// TIA Portal project "Blister 080520_V16_1" (V16)

(* hardware
DEVICE "S7-1200 station_1"  S7-1200 Station
   slot 0: "Rack_0"  S7-1200 Rack  Rack  V1.0
   slot 1: "PLC_1"  CPU 1215C DC/DC/DC  6ES7 215-1AG40-0XB0  V4.2
DEVICE "PC-System_1"  SIMATIC PC station
   slot 0: "SIMATIC PC station"  Rail  SIMATIC PC-Station  V1.0
      slot 125: "Stationmanager"  Station_Manager  V6.0.4
   slot 1: "HMI_RT_1"  WinCC RT Advanced  6AV2 104-0xxxx-xxxx  15.0.0.0
      slot 33792: "Host interface"  Host interface
   slot 2: "IE general_1"  IE General  IE_CP  V8.2.0
*)

// ===== PLC "PLC_1"  CPU 1215C DC/DC/DC =====

VAR_GLOBAL   // PLC tag table "Default tag table"
   "System_Byte" AT %MB1000 : Byte;
   "FirstScan" AT %M1000.0 : Bool;
   "DiagStatusUpdate" AT %M1000.1 : Bool;
   "AlwaysTRUE" AT %M1000.2 : Bool;
   "AlwaysFALSE" AT %M1000.3 : Bool;
   "Clock_Byte" AT %MB1001 : Byte;
   "Clock_10Hz" AT %M1001.0 : Bool;
   "Clock_5Hz" AT %M1001.1 : Bool;
   "Clock_2.5Hz" AT %M1001.2 : Bool;
   "Clock_2Hz" AT %M1001.3 : Bool;
   "Clock_1.25Hz" AT %M1001.4 : Bool;
   "Clock_1Hz" AT %M1001.5 : Bool;
   "Clock_0.625Hz" AT %M1001.6 : Bool;
   "Clock_0.5Hz" AT %M1001.7 : Bool;
   "System_Byte(1)" AT %MB1000 : Byte;
   "point_1" AT %M0.0 : Bool;
   "point_2" AT %M0.1 : Bool;
   "a" AT %MD2 : Real;
   "e" AT %MD6 : Real;
   "g" AT %MD10 : Real;
   "ii" AT %MD14 : Real;
   "oo" AT %MD18 : Real;
   "pp" AT %MD22 : Real;
   "rr" AT %MD26 : Real;
   "Run" AT %M0.2 : Bool;
   "Shift" AT %M0.3 : Bool;
   "Trig_2" AT %M0.4 : Bool;
   "Enable" AT %M0.5 : Bool;
   "Timer_Main" AT %MD30 : Time;
   "Angle" AT %MW34 : Int;
   "Temp_1" AT %MD44 : Real;
   "Forming_Trig" AT %M0.6 : Bool;
   "Forming_Enable" AT %M0.7 : Bool;
   "Servo_Pull_Enable" AT %M1.0 : Bool;
   "Servo_Pull_CCW_Trig" AT %M1.1 : Bool;
   "Servo_Pull_CW_Trig" AT %M1.2 : Bool;
   "PinHole_Detect" AT %M1.3 : Bool;
   "Trig3" AT %M1.4 : Bool;
   "PinHole_Write" AT %M1.5 : Bool;
   "T_Simu_Angle" AT %MW36 : Int;
   "Simu_Angle_2" AT %MD38 : Time;
   "Trig4" AT %M1.6 : Bool;
   "Trig5" AT %M1.7 : Bool;
   "Reset_C" AT %M42.0 : Bool;
   "Trig6" AT %M42.1 : Bool;
   "Step" AT %MW52 : Int;
   "EN_Feed_1_Step" AT %M42.2 : Bool;
   "Feeder_Enough_Step" AT %M42.3 : Bool;
   "Trig8" AT %M42.4 : Bool;
   "Set" AT %M42.5 : Bool;
   "Trig9" AT %M42.6 : Bool;
   "Do" AT %M42.7 : Bool;
   "Trig11" AT %M43.0 : Bool;
   "trig12" AT %M43.1 : Bool;
   "Feeder_Trig" AT %M43.2 : Bool;
   "Feeder_Enough_Angle" AT %M43.3 : Bool;
   "Step_Calcu" AT %MW48 : Int;
   "Trig13" AT %M43.4 : Bool;
   "Pull_2" AT %M43.5 : Bool;
   "trig14" AT %M43.6 : Bool;
   "trig15" AT %M43.7 : Bool;
   "trig16" AT %M50.0 : Bool;
   "Ghi" AT %M50.1 : Bool;
   "Ghi2" AT %M50.2 : Bool;
   "Write_not_feed" AT %M50.3 : Bool;
   "Trig17" AT %M50.4 : Bool;
   "Write_not_feed_2" AT %M50.5 : Bool;
   "trig18" AT %M50.6 : Bool;
   "Write_feed_ok" AT %M50.7 : Bool;
   "Write_not_feed_3" AT %M51.0 : Bool;
   "test" AT %M51.1 : Bool;
   "testmw" AT %MB54 : Byte;
END_VAR

DATA_BLOCK "Forming_Aplice_DB"   // DB9
{ S7_Optimized_Access := 'TRUE' }
VERSION : 0.1
// stored: InstanceOfName Forming_Aplice
"Forming_Aplice"
BEGIN
END_DATA_BLOCK

DATA_BLOCK "Blister_Animation"   // DB10
{ S7_Optimized_Access := 'TRUE' }
VERSION : 0.1
   VAR
      Blister_1 : Array[0..50] of Word;
      Blister_Matrix : Array[0..50] of Word;
   END_VAR
BEGIN
END_DATA_BLOCK

DATA_BLOCK "Blister_Show"   // DB11
{ S7_Optimized_Access := 'TRUE' }
VERSION : 0.1
   VAR RETAIN
      Total_Row : Int := 6;
      Total_Blister_Column : Int := 20;
   END_VAR
   VAR
      Total_Blister_Column_Temp : Int := 20;
      Arr : Array[0..10] of Int;
   END_VAR
BEGIN
END_DATA_BLOCK

DATA_BLOCK "Shift_Blister_DB"   // DB12
{ S7_Optimized_Access := 'TRUE' }
VERSION : 0.1
// stored: InstanceOfName Shift_Blister
"Shift_Blister"
BEGIN
END_DATA_BLOCK

DATA_BLOCK "Station_Position"   // DB13
{ S7_Optimized_Access := 'TRUE' }
VERSION : 0.1
   VAR
      Cut_to_ApliceALU : Int := 5;
      Cut_to_Camera : Int := 8;
      Cut_to_Matrix_Feeder : Int := 11;
      Cut_to_PinHole : Int := 14;
      Cut_to_Forming : Int := 17;
   END_VAR
BEGIN
END_DATA_BLOCK

DATA_BLOCK "Machine_Data"   // DB14
{ S7_Optimized_Access := 'TRUE' }
VERSION : 0.1
   VAR RETAIN
      Angle : Int;
      Length_Step : Int := 83;
      SV_Machine_Speed : Int := 30;
   END_VAR
BEGIN
END_DATA_BLOCK

DATA_BLOCK "Matrix_Feeder_DB"   // DB15
{ S7_Optimized_Access := 'TRUE' }
VERSION : 0.1
// stored: InstanceOfName Matrix_Feeder
"Matrix_Feeder"
BEGIN
END_DATA_BLOCK

DATA_BLOCK "Write_Blister_Animation_DB"   // DB17
{ S7_Optimized_Access := 'TRUE' }
VERSION : 0.1
// stored: InstanceOfName Write_Blister_Animation
"Write_Blister_Animation"
BEGIN
END_DATA_BLOCK

DATA_BLOCK "Forming_Module_DB"   // DB20
{ S7_Optimized_Access := 'TRUE' }
VERSION : 0.1
// stored: InstanceOfName Forming_Module
"Forming_Module"
BEGIN
END_DATA_BLOCK

DATA_BLOCK "Batch_Management_DB"   // DB22
{ S7_Optimized_Access := 'TRUE' }
VERSION : 0.1
// stored: InstanceOfName Batch_Management
"Batch_Management"
BEGIN
   Lot_Size := 500;
   SV_Sampling_Time := 1;
   Q_Reset_New_Lot := TRUE;
   Reset_Sampling_Time := TRUE;
   C1.QD := TRUE;
   C1.PV := 100000;
   T_Sampling_Time_1.ST := T#52M_54S_448MS;
   T_Sampling_Time_2.ST := T#52M_54S_448MS;
   T.ST := T#52M_54S_448MS;
   T.PT := T#1M_40S;
END_DATA_BLOCK

DATA_BLOCK "Total_Time_Run_DB"   // DB23
{ S7_Optimized_Access := 'TRUE' }
VERSION : 0.1
// stored: InstanceOfName Total_Time_Run
"Total_Time_Run"
BEGIN
END_DATA_BLOCK

DATA_BLOCK "Recipe_Data"   // DB24
{ S7_Optimized_Access := 'TRUE' }
VERSION : 0.1
   VAR RETAIN
      Data_1 : Int;
      Data_2 : Int;
      Data_3 : Int;
      Data_4 : Int;
      Data_5 : Int;
   END_VAR
BEGIN
END_DATA_BLOCK

DATA_BLOCK "Batch_Data"   // DB25
{ S7_Optimized_Access := 'TRUE' }
VERSION : 0.1
   VAR RETAIN
      Time_Start : DTL;
      Time_Stop : DTL;
   END_VAR
BEGIN
END_DATA_BLOCK

// folder: DB_of_FB

DATA_BLOCK "Calib_Speed_DB"   // DB1
{ S7_Optimized_Access := 'TRUE' }
VERSION : 0.1
// stored: InstanceOfName Calib_Speed_Output
"Calib_Speed_Output"
BEGIN
END_DATA_BLOCK

DATA_BLOCK "Scale_Analog_DB"   // DB3
{ S7_Optimized_Access := 'TRUE' }
VERSION : 0.1
// stored: InstanceOfName Scale_Analog_Output
"Scale_Analog_Output"
BEGIN
END_DATA_BLOCK

DATA_BLOCK "Scale_Analog_Input_DB"   // DB4
{ S7_Optimized_Access := 'TRUE' }
VERSION : 0.1
// stored: InstanceOfName Scale_Analog_Input
"Scale_Analog_Input"
BEGIN
END_DATA_BLOCK

DATA_BLOCK "Calib_Temperature_Input_DB"   // DB5
{ S7_Optimized_Access := 'TRUE' }
VERSION : 0.1
// stored: InstanceOfName Calib_Temperature_Input
"Calib_Temperature_Input"
BEGIN
END_DATA_BLOCK

// folder: Main_program/Conveyor

DATA_BLOCK "Conveyor"   // DB2
{ S7_Optimized_Access := 'TRUE' }
VERSION : 0.1
   VAR
      Calib_Enable : Bool;
      B_Calib_Dim_Point_1 : Bool;
      B_Calib_Dim_Point_2 : Bool;
      SV_Calib_Speed_Point_1 : Int;
      SV_Calib_Speed_Point_2 : Int;
   END_VAR
   VAR RETAIN
      Calib_Range_Analog_Low : Int;
      Calib_Range_Analog_High : Int;
      Calib_Range_Speed_Low : Int;
      Calib_Range_Speed_High : Int;
   END_VAR
   VAR
      SV_Speed : Int;
      O_Analog : Int;
      B_RunConveyor_Speed_Min : Bool;
      B_RunConveyor_Speed_Max : Bool;
      B_Calib_OK : Bool;
      B_Calib_Default : Bool;
      O_Calib_Result : Bool;
      O_Run : Bool;
      H_PID_State : Int;
      H_Stop_Kp : Real;
      H_Stop_Ki : Real;
      H_Stop_Kd : Real;
      H_Run_Kp : Real;
      H_Run_Ki : Real;
      H_Run_Kd : Real;
      B_PID_Default : Bool;
      Stop_Kp_1 : Real;
      Stop_Ki_1 : Real;
      Stop_Kd_1 : Real;
      Run_Kp_1 : Real;
      Run_Ki_1 : Real;
      Run_Kd_1 : Real;
   END_VAR
BEGIN
END_DATA_BLOCK

DATA_BLOCK "PID Setting_DB"   // DB8
{ S7_Optimized_Access := 'TRUE' }
VERSION : 0.1
// stored: InstanceOfName PID Setting
"PID Setting"
BEGIN
END_DATA_BLOCK

// folder: Main_program/Temperature_Top

DATA_BLOCK "Temperature_Top"   // DB6
{ S7_Optimized_Access := 'TRUE' }
VERSION : 0.1
   VAR
      Calib_Enable : Bool;
      B_Calib_Dim_Point_1 : Bool;
      B_Calib_Dim_Point_2 : Bool;
   END_VAR
   VAR RETAIN
      O_Calib_Range_Analog_Min : Int;
      O_Calib_Range_Analog_Max : Int;
      O_Calib_Range_Temper_Min : Int;
      O_Calib_Range_Temper_Max : Int;
   END_VAR
   VAR
      PV_Temper : Int;
      B_Calib_OK : Bool;
      B_Default : Bool;
      I_Analog_Read : Int;
      B_Default_3 : Bool;
      Calib_Result : Bool;
      SV_Point_1_Temper : Int;
      SV_Point_2_Temper : Int;
      SV_Temper : Int;
      PWM_Out : Bool;
   END_VAR
BEGIN
END_DATA_BLOCK

// folder: System blocks/Program resources

DATA_BLOCK "IEC_Timer_0_DB"   // DB16
{ S7_Optimized_Access := 'TRUE' }
AUTHOR : Simatic
FAMILY : IEC
NAME : IEC_TMR
VERSION : 1.0
// stored: InstanceOfName IEC_TIMER
"IEC_TIMER"
BEGIN
END_DATA_BLOCK

DATA_BLOCK "IEC_Timer_0_DB_1"   // DB18
{ S7_Optimized_Access := 'TRUE' }
AUTHOR : Simatic
FAMILY : IEC
NAME : IEC_TMR
VERSION : 1.0
// stored: InstanceOfName IEC_TIMER
"IEC_TIMER"
BEGIN
END_DATA_BLOCK

DATA_BLOCK "IEC_Timer_0_DB_2"   // DB19
{ S7_Optimized_Access := 'TRUE' }
AUTHOR : Simatic
FAMILY : IEC
NAME : IEC_TMR
VERSION : 1.0
// stored: InstanceOfName IEC_TIMER
"IEC_TIMER"
BEGIN
END_DATA_BLOCK

DATA_BLOCK "IEC_Timer_0_DB_3"   // DB21
{ S7_Optimized_Access := 'TRUE' }
AUTHOR : Simatic
FAMILY : IEC
NAME : IEC_TMR
VERSION : 1.0
// stored: InstanceOfName IEC_TIMER
"IEC_TIMER"
BEGIN
END_DATA_BLOCK

// folder: (top level)

FUNCTION_BLOCK "Forming_Aplice"   // FB6, LAD
{ S7_Optimized_Access := 'TRUE' }
VERSION : 0.1
   VAR_INPUT
      Sensor : Bool;
   END_VAR
BEGIN

REGION Network 1
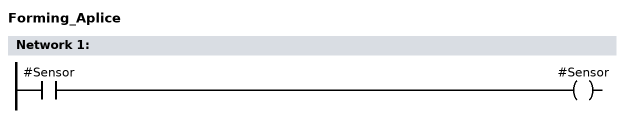
   RUNG wire#powerrail
      Contact( #Sensor )
      Coil( #Sensor )
   END_RUNG
   // the same network as SCL:
   #Sensor := #Sensor;
END_REGION
END_FUNCTION_BLOCK

FUNCTION_BLOCK "Shift_Blister"   // FB7, LAD
{ S7_Optimized_Access := 'TRUE' }
VERSION : 0.1
   VAR_INPUT
      Number_Column : Int;
   END_VAR
   VAR_IN_OUT
      Trig : Bool;
   END_VAR
   VAR
      i : Int;
   END_VAR
BEGIN

REGION Network 2 (SCL)
   IF #Trig = TRUE THEN
       "Blister_Animation".Blister_1[#Number_Column + 1] := 0;
       FOR #i := 0 TO #Number_Column DO
           "Blister_Animation".Blister_1[#i] := "Blister_Animation".Blister_1[#i + 1];
           "Blister_Animation".Blister_Matrix[#i] := "Blister_Animation".Blister_Matrix[#i + 1];
       END_FOR;
       #Trig := FALSE;
       // #Do := FALSE;
   END_IF;
END_REGION
END_FUNCTION_BLOCK

FUNCTION_BLOCK "Matrix_Feeder"   // FB8, LAD
{ S7_Optimized_Access := 'TRUE' }
VERSION : 0.1
   VAR_INPUT
      Angel_Machine : Int;
      Pull_Trig : Bool;
      "Switch_on/off" : Bool;
   END_VAR
   VAR_OUTPUT
      Q_Feeder : Bool;
   END_VAR
   VAR
      Counte : IEC_COUNTER;
   END_VAR
   VAR RETAIN
      Feed_1_Step : Bool;
      EN_Feed_2_Step : Bool;
   END_VAR
   VAR
      Feed_2_Step : Bool;
      Angel_Begin : Int := 170;
      Angel_End : Int := 210;
      Angel_Begin_Offset : Int;
      I_Step_Feeder : Int := 1;
      Trig1 : Bool;
   END_VAR
   VAR_TEMP   // added for the SCL form of the ladder/FBD networks
      _w1 : Bool;
      _w2 : Bool;
   END_VAR
BEGIN

REGION Network 1: Reset step feer
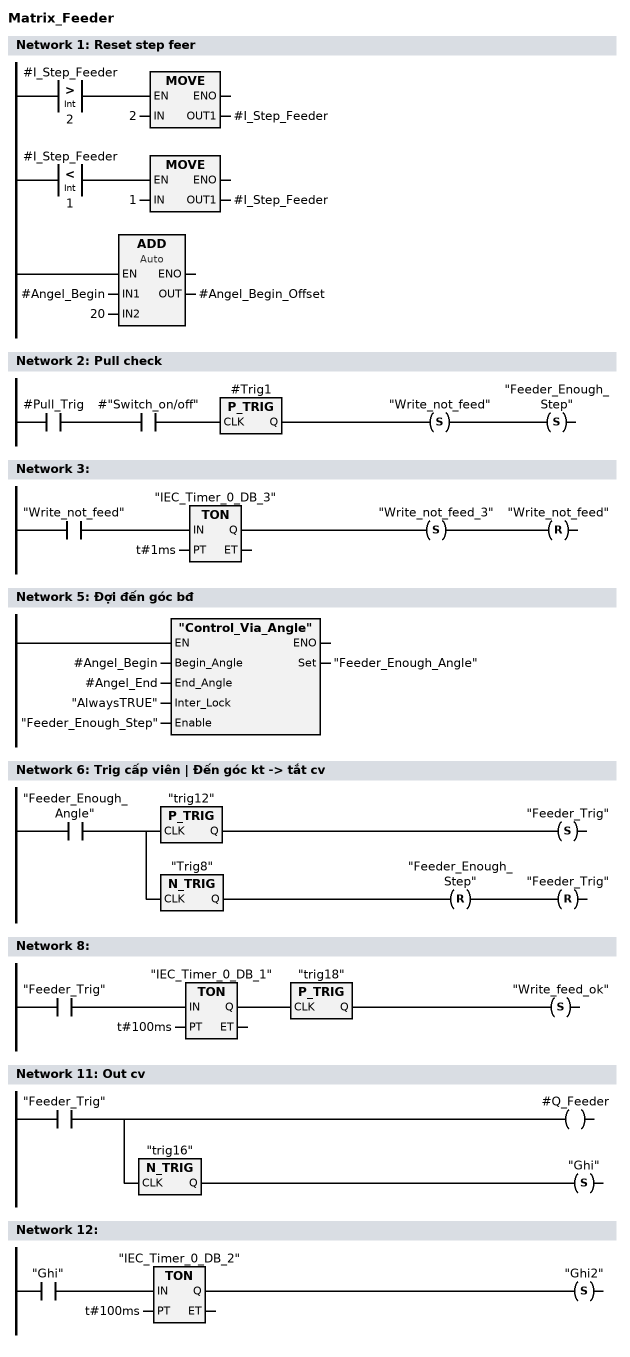
   RUNG wire#powerrail
      { S7_Templates := "SrcType := Int" } GT_Contact(in1 := #I_Step_Feeder, in2 := 2)
      Move(in := 2, out1 => #I_Step_Feeder)
   END_RUNG
   RUNG wire#powerrail
      { S7_Templates := "SrcType := Int" } LT_Contact(in1 := #I_Step_Feeder, in2 := 1)
      Move(in := 1, out1 => #I_Step_Feeder)
   END_RUNG
   RUNG wire#powerrail
      Add(in1 := #Angel_Begin, in2 := 20, out => #Angel_Begin_Offset)
   END_RUNG
   // the same network as SCL:
   IF #I_Step_Feeder > 2 THEN #I_Step_Feeder := 2; END_IF;
   IF #I_Step_Feeder < 1 THEN #I_Step_Feeder := 1; END_IF;
   #Angel_Begin_Offset := #Angel_Begin + 20;
END_REGION

REGION Network 2: Pull check
   RUNG wire#powerrail
      Contact( #Pull_Trig )
      Contact( #"Switch_on/off" )
      P_Trig( #Trig1 )
      S_Coil( "Write_not_feed" )
      S_Coil( "Feeder_Enough_Step" )
   END_RUNG
   // the same network as SCL:
   #_w1 := #Pull_Trig AND #"Switch_on/off";
   #_w2 := #_w1 AND NOT #Trig1;   // rising edge
   #Trig1 := #_w1;
   IF #_w2 THEN
       "Write_not_feed" := TRUE;
       "Feeder_Enough_Step" := TRUE;
   END_IF;
END_REGION

REGION Network 3
   "IEC_Timer_0_DB_3".TON(IN := "Write_not_feed", PT := t#1ms);
   IF "IEC_Timer_0_DB_3".Q THEN
       "Write_not_feed_3" := TRUE;
       "Write_not_feed" := FALSE;
   END_IF;
END_REGION

REGION Network 4 (SCL)
   //IF FALSE = true THEN
   IF "Write_not_feed_3" = true THEN
       //  Bước cv = 2 thi kiem tra 2 hang
       IF #I_Step_Feeder = 2 THEN
           "Blister_Animation".Blister_1["Station_Position".Cut_to_Matrix_Feeder] := 0;
           "Blister_Animation".Blister_1["Station_Position".Cut_to_Matrix_Feeder + 1] := 0;
       END_IF;
       // = 1
       IF #I_Step_Feeder = 1 THEN
           "Blister_Animation".Blister_1["Station_Position".Cut_to_Matrix_Feeder] := 0;
       END_IF;
       "Write_not_feed_3" := FALSE;
   END_IF;
END_REGION

REGION Network 5: Đợi đến góc bđ
   RUNG wire#powerrail
      "Control_Via_Angle"(Begin_Angle := #Angel_Begin, End_Angle := #Angel_End, Inter_Lock := "AlwaysTRUE", Enable := "Feeder_Enough_Step", Set => "Feeder_Enough_Angle")
   END_RUNG
   // the same network as SCL:
   "Control_Via_Angle"(Begin_Angle := #Angel_Begin,
                       End_Angle := #Angel_End,
                       Inter_Lock := "AlwaysTRUE",
                       Enable := "Feeder_Enough_Step",
                       Set => "Feeder_Enough_Angle");
END_REGION

REGION Network 6: Trig cấp viên | Đến góc kt -> tắt cv
   RUNG wire#powerrail
      Contact( "Feeder_Enough_Angle" )
      wire#w1
      P_Trig( "trig12" )
      S_Coil( "Feeder_Trig" )
   END_RUNG
   RUNG wire#w1
      N_Trig( "Trig8" )
      R_Coil( "Feeder_Enough_Step" )
      R_Coil( "Feeder_Trig" )
   END_RUNG
   // the same network as SCL:
   #_w1 := "Feeder_Enough_Angle" AND NOT "trig12";   // rising edge
   "trig12" := "Feeder_Enough_Angle";
   IF #_w1 THEN "Feeder_Trig" := TRUE; END_IF;
   #_w2 := NOT "Feeder_Enough_Angle" AND "Trig8";   // falling edge
   "Trig8" := "Feeder_Enough_Angle";
   IF #_w2 THEN
       "Feeder_Enough_Step" := FALSE;
       "Feeder_Trig" := FALSE;
   END_IF;
END_REGION

REGION Network 7 (SCL): Kiểm tra đk cv | buoc cv = 1 or 2
   //IF FALSE = true THEN
   IF "Feeder_Trig" = true THEN
      //  Bước cv = 2 thi kiem tra 2 hang
       IF #I_Step_Feeder = 2 THEN 
           IF "Blister_Animation".Blister_Matrix["Station_Position".Cut_to_Matrix_Feeder] <> 16#3F OR "Blister_Animation".Blister_Matrix["Station_Position".Cut_to_Matrix_Feeder + 1] <> 16#3F THEN
               "Feeder_Trig" := FALSE;
           END_IF;
      END_IF;
       // = 1
       IF #I_Step_Feeder = 1 THEN
           IF "Blister_Animation".Blister_Matrix["Station_Position".Cut_to_Matrix_Feeder] <> 16#3F THEN
               "Feeder_Trig" := FALSE;
               "Blister_Animation".Blister_1["Station_Position".Cut_to_Matrix_Feeder] := 0;
           END_IF;
       END_IF;
   END_IF;
END_REGION

REGION Network 8
   "IEC_Timer_0_DB_1".TON(IN := "Feeder_Trig", PT := t#100ms);
   #_w1 := "IEC_Timer_0_DB_1".Q AND NOT "trig18";   // rising edge
   "trig18" := "IEC_Timer_0_DB_1".Q;
   IF #_w1 THEN "Write_feed_ok" := TRUE; END_IF;
END_REGION

REGION Network 9 (SCL)
   //IF FALSE = true THEN
   IF "Write_feed_ok" = true THEN
       //  Bước cv = 2 thi ghi 2 hang ok sau khi qua cvmt
       IF #I_Step_Feeder = 2 THEN
           "Blister_Animation".Blister_1["Station_Position".Cut_to_Matrix_Feeder] := 16#3f;
           "Blister_Animation".Blister_1["Station_Position".Cut_to_Matrix_Feeder + 1] := 16#3f;
       END_IF;
       // = 1
       IF #I_Step_Feeder = 1 THEN
           "Blister_Animation".Blister_1["Station_Position".Cut_to_Matrix_Feeder] := 16#3f;
       END_IF;
       "Write_feed_ok" := FALSE;
   END_IF;
END_REGION

REGION Network 10 (SCL)
   IF "Write_not_feed_2" = TRUE THEN
       "Blister_Animation".Blister_1["Station_Position".Cut_to_Matrix_Feeder] := 0;
       "Blister_Animation".Blister_1["Station_Position".Cut_to_Matrix_Feeder + 1] := 0;
       ;
   "Write_not_feed_2" := FALSE;
   END_IF;
END_REGION

REGION Network 11: Out cv
   RUNG wire#powerrail
      Contact( "Feeder_Trig" )
      wire#w1
      Coil( #Q_Feeder )
   END_RUNG
   RUNG wire#w1
      N_Trig( "trig16" )
      S_Coil( "Ghi" )
   END_RUNG
   // the same network as SCL:
   #Q_Feeder := "Feeder_Trig";
   #_w1 := NOT "Feeder_Trig" AND "trig16";   // falling edge
   "trig16" := "Feeder_Trig";
   IF #_w1 THEN "Ghi" := TRUE; END_IF;
END_REGION

REGION Network 12
   "IEC_Timer_0_DB_2".TON(IN := "Ghi", PT := t#100ms);
   IF "IEC_Timer_0_DB_2".Q THEN "Ghi2" := TRUE; END_IF;
END_REGION

REGION Network 13 (SCL): Ghi gia tri 0 sau khi cap vien ok
   IF "Ghi2" = true THEN
       IF #I_Step_Feeder = 2 THEN
           "Blister_Animation".Blister_Matrix["Station_Position".Cut_to_Matrix_Feeder] := 0;
           "Blister_Animation".Blister_Matrix["Station_Position".Cut_to_Matrix_Feeder + 1] := 0;
           ;
       END_IF;
       // buoc cv = 1
       IF #I_Step_Feeder = 1 THEN
           "Blister_Animation".Blister_Matrix["Station_Position".Cut_to_Matrix_Feeder] := 0;
           ;
       END_IF;
   "Ghi" := FALSE;
   "Ghi2" := FALSE;
   END_IF;
END_REGION
END_FUNCTION_BLOCK

FUNCTION_BLOCK "Write_Blister_Animation"   // FB9, LAD
{ S7_Optimized_Access := 'TRUE' }
VERSION : 0.1
   VAR_INPUT
      Forming_Trig : Bool;
   END_VAR
   VAR
      Trig : Bool;
      Write_Forming : Bool;
   END_VAR
   VAR_TEMP   // added for the SCL form of the ladder/FBD networks
      _w1 : Bool;
   END_VAR
BEGIN

REGION Network 1
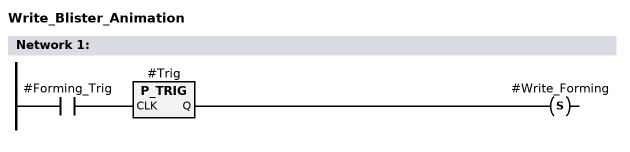
   RUNG wire#powerrail
      Contact( #Forming_Trig )
      P_Trig( #Trig )
      S_Coil( #Write_Forming )
   END_RUNG
   // the same network as SCL:
   #_w1 := #Forming_Trig AND NOT #Trig;   // rising edge
   #Trig := #Forming_Trig;
   IF #_w1 THEN #Write_Forming := TRUE; END_IF;
END_REGION

REGION Network 2 (SCL)
   IF #Write_Forming = TRUE THEN
       "Blister_Animation".Blister_1["Station_Position".Cut_to_Forming] := 2#111111;
       "Blister_Animation".Blister_Matrix["Station_Position".Cut_to_Forming] := 2#111111;
       #Write_Forming := FALSE;

   END_IF;
END_REGION
END_FUNCTION_BLOCK

FUNCTION_BLOCK "Forming_Module"   // FB10, LAD
{ S7_Optimized_Access := 'TRUE' }
VERSION : 0.1
   VAR_INPUT
      Inter_Lock : Bool;
   END_VAR
   VAR_OUTPUT
      Forming_Trig : Bool;
   END_VAR
   VAR RETAIN
      SV_Angle_Forming_Begin : Int := 160;
      SV_Angle_Forming_End : Int := 200;
   END_VAR
   VAR
      Forming_Switch : Bool;
   END_VAR
BEGIN

REGION Network 1
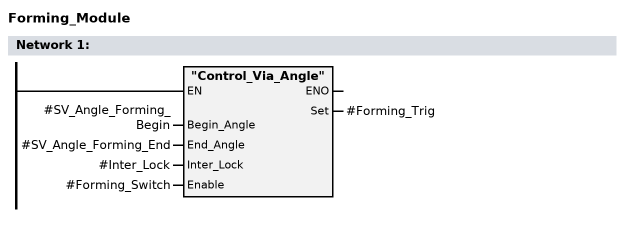
   RUNG wire#powerrail
      "Control_Via_Angle"(Begin_Angle := #SV_Angle_Forming_Begin, End_Angle := #SV_Angle_Forming_End, Enable := #Forming_Switch, Inter_Lock := #Inter_Lock, Set => #Forming_Trig)
   END_RUNG
   // the same network as SCL:
   "Control_Via_Angle"(Begin_Angle := #SV_Angle_Forming_Begin,
                       End_Angle := #SV_Angle_Forming_End,
                       Inter_Lock := #Inter_Lock,
                       Enable := #Forming_Switch,
                       Set => #Forming_Trig);
END_REGION
END_FUNCTION_BLOCK

FUNCTION_BLOCK "Batch_Management"   // FB11, LAD
{ S7_Optimized_Access := 'TRUE' }
VERSION : 0.1
   VAR_INPUT
      I_Machine_Run : Bool;
      Lot_Size : DInt;
      SV_Sampling_Time : DInt;
      Product_Name : Int;
      Batch_Number : Int;
      Batch_Size : DInt;
   END_VAR
   VAR_OUTPUT
      Q_Write_Report : Bool;
   END_VAR
   VAR_IN_OUT
      B_Start_Lot : Bool;
      B_Finish_Lot : Bool;
      B_Hold_Lot : Bool;
      Q_Reset_New_Lot : Bool;
      Reset_Sampling_Time : Bool;
      PV_Lot_Start_Time : DTL;
      PV_Lot_End_Time : DTL;
      PV_Lot_Status : USInt := 0;
      PV_Lot_Running_Total_Time : DInt;
   END_VAR
   VAR
      Trig : Bool;
      Trig2 : Bool;
      Trig3 : Bool;
      Trig4 : Bool;
      RET_VAL_1 : Int;
      RET_VAL_2 : Int;
      C1 : IEC_DCOUNTER;
   END_VAR
   VAR RETAIN
      T_Sampling_Time_1 : IEC_TIMER;
   END_VAR
   VAR
      T_Sampling_Time_2 : IEC_TIMER;
      PV_Sampling_Time : DInt;
      Trig5 : Bool;
      T : IEC_TIMER;
      Recipe_Name_1 : String;
      Recipe_Name_2 : String;
      Recipe_Record_1 : Int;
      Recipe_Record_2 : Int;
      Record_Number : Int;
   END_VAR
   VAR CONSTANT
      Running : USInt := 2;
      Finish : USInt := 0;
      Holding : USInt := 1;
   END_VAR
   VAR_TEMP   // added for the SCL form of the ladder/FBD networks
      _w1 : Bool;
      _w2 : Bool;
      _w3 : Bool;
      _w4 : Bool;
   END_VAR
BEGIN

REGION Network 1: Thời điểm bắt đầu lô
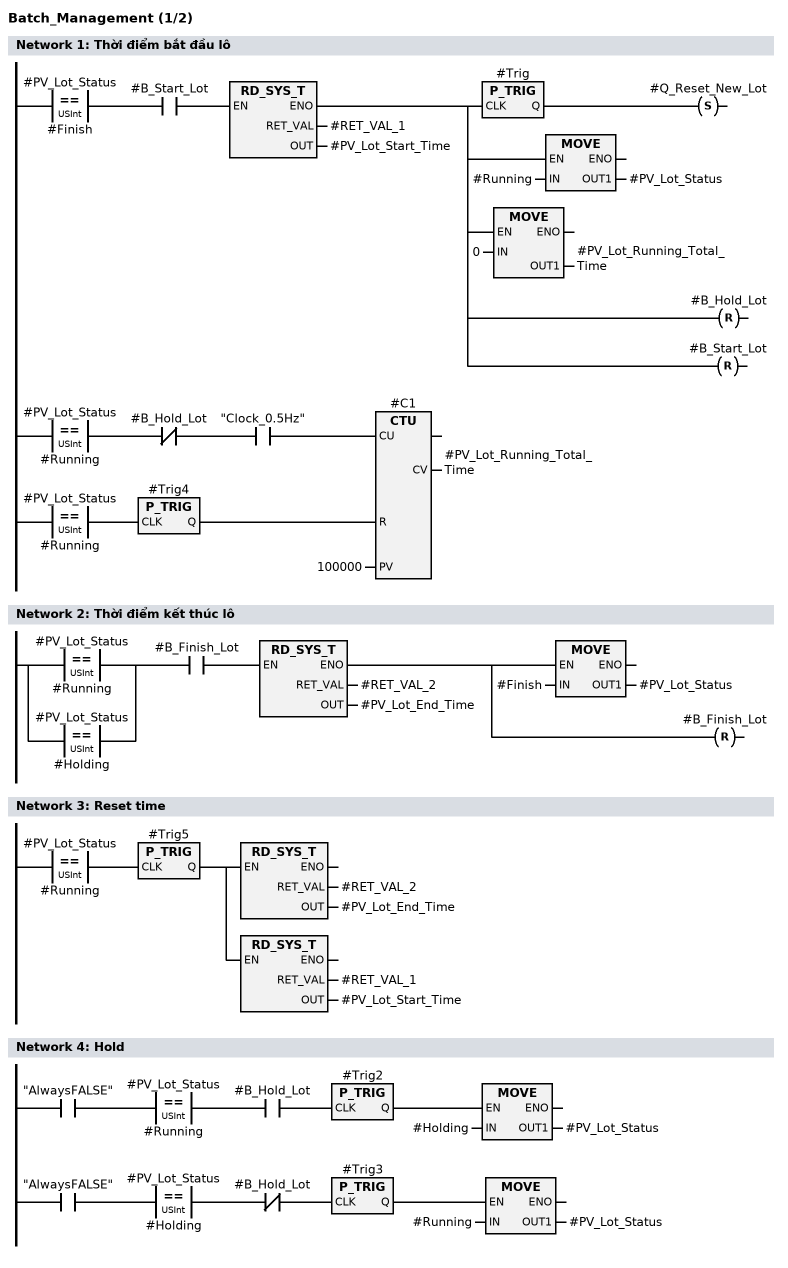
   // ENO of a box is taken as its EN; it also drops when the box reports an error
   #_w1 := (#PV_Lot_Status = #Finish) AND #B_Start_Lot;
   IF #_w1 THEN #RET_VAL_1 := RD_SYS_T(OUT => #PV_Lot_Start_Time); END_IF;
   #_w2 := #_w1 AND NOT #Trig;   // rising edge
   #Trig := #_w1;
   IF #_w2 THEN #Q_Reset_New_Lot := TRUE; END_IF;
   IF #_w1 THEN
       #PV_Lot_Status := #Running;
       #PV_Lot_Running_Total_Time := 0;
       #B_Hold_Lot := FALSE;
       #B_Start_Lot := FALSE;
   END_IF;
   #_w3 := #PV_Lot_Status = #Running;
   #_w4 := #_w3 AND NOT #Trig4;   // rising edge
   #Trig4 := #_w3;
   #C1.CTU(CU := (#PV_Lot_Status = #Running) AND NOT #B_Hold_Lot AND "Clock_0.5Hz",
           R := #_w4,
           PV := 100000,
           CV => #PV_Lot_Running_Total_Time);
END_REGION

REGION Network 2: Thời điểm kết thúc lô
   // ENO of a box is taken as its EN; it also drops when the box reports an error
   IF ((#PV_Lot_Status = #Running) OR (#PV_Lot_Status = #Holding)) AND #B_Finish_Lot THEN
       #RET_VAL_2 := RD_SYS_T(OUT => #PV_Lot_End_Time);
   END_IF;
   #_w1 := ((#PV_Lot_Status = #Running) OR (#PV_Lot_Status = #Holding)) AND #B_Finish_Lot;
   IF #_w1 THEN
       #PV_Lot_Status := #Finish;
       #B_Finish_Lot := FALSE;
   END_IF;
END_REGION

REGION Network 3: Reset time
   #_w1 := #PV_Lot_Status = #Running;
   #_w2 := #_w1 AND NOT #Trig5;   // rising edge
   #Trig5 := #_w1;
   IF #_w2 THEN
       #RET_VAL_2 := RD_SYS_T(OUT => #PV_Lot_End_Time);
       #RET_VAL_1 := RD_SYS_T(OUT => #PV_Lot_Start_Time);
   END_IF;
END_REGION

REGION Network 4: Hold
   RUNG wire#powerrail
      Contact( "AlwaysFALSE" )
      { S7_Templates := "SrcType := USInt" } EQ_Contact(in1 := #PV_Lot_Status, in2 := #Running)
      Contact( #B_Hold_Lot )
      P_Trig( #Trig2 )
      Move(in := #Holding, out1 => #PV_Lot_Status)
   END_RUNG
   RUNG wire#powerrail
      Contact( "AlwaysFALSE" )
      { S7_Templates := "SrcType := USInt" } EQ_Contact(in1 := #PV_Lot_Status, in2 := #Holding)
      I_Contact( #B_Hold_Lot )
      P_Trig( #Trig3 )
      Move(in := #Running, out1 => #PV_Lot_Status)
   END_RUNG
   // the same network as SCL:
   #_w1 := "AlwaysFALSE" AND (#PV_Lot_Status = #Running) AND #B_Hold_Lot;
   #_w2 := #_w1 AND NOT #Trig2;   // rising edge
   #Trig2 := #_w1;
   IF #_w2 THEN #PV_Lot_Status := #Holding; END_IF;
   #_w3 := "AlwaysFALSE" AND (#PV_Lot_Status = #Holding) AND NOT #B_Hold_Lot;
   #_w4 := #_w3 AND NOT #Trig3;   // rising edge
   #Trig3 := #_w3;
   IF #_w4 THEN #PV_Lot_Status := #Running; END_IF;
END_REGION

REGION Network 5: Write report
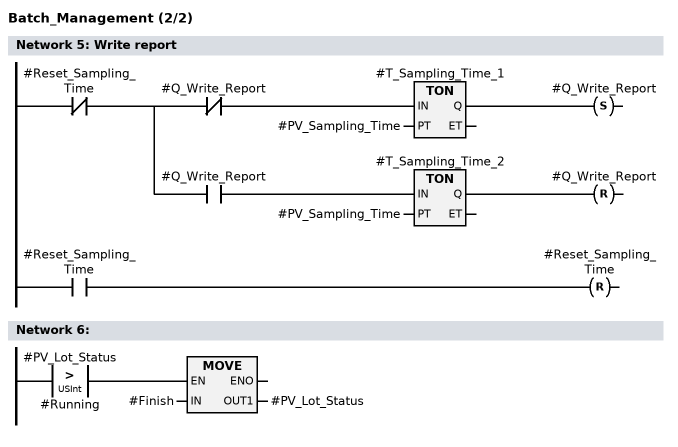
   #T_Sampling_Time_1.TON(IN := NOT #Reset_Sampling_Time AND NOT #Q_Write_Report, PT := #PV_Sampling_Time);
   IF #T_Sampling_Time_1.Q THEN #Q_Write_Report := TRUE; END_IF;
   #T_Sampling_Time_2.TON(IN := NOT #Reset_Sampling_Time AND #Q_Write_Report, PT := #PV_Sampling_Time);
   IF #T_Sampling_Time_2.Q THEN #Q_Write_Report := FALSE; END_IF;
   IF #Reset_Sampling_Time THEN #Reset_Sampling_Time := FALSE; END_IF;
END_REGION

REGION Network 6
   RUNG wire#powerrail
      { S7_Templates := "SrcType := USInt" } GT_Contact(in1 := #PV_Lot_Status, in2 := #Running)
      Move(in := #Finish, out1 => #PV_Lot_Status)
   END_RUNG
   // the same network as SCL:
   IF #PV_Lot_Status > #Running THEN #PV_Lot_Status := #Finish; END_IF;
END_REGION
END_FUNCTION_BLOCK

FUNCTION_BLOCK "Total_Time_Run"   // FB12, LAD
{ S7_Optimized_Access := 'TRUE' }
VERSION : 0.1
   VAR_OUTPUT
      "PV_Total_Time_Run_(s)" : DInt;
   END_VAR
   VAR
      C1 : IEC_DCOUNTER;
   END_VAR
BEGIN

REGION Network 1
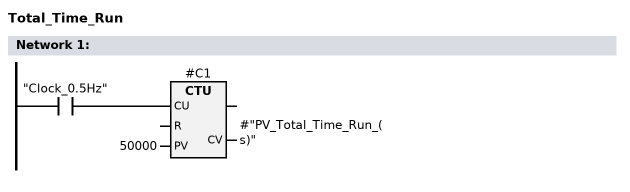
   #C1.CTU(CU := "Clock_0.5Hz", PV := 50000, CV => #"PV_Total_Time_Run_(s)");
END_REGION
END_FUNCTION_BLOCK

FUNCTION "Angle_Simu" : Void   // FC6, LAD
{ S7_Optimized_Access := 'TRUE' }
VERSION : 0.1
   VAR_TEMP
      RS : Bool;
   END_VAR
BEGIN

REGION Network 1
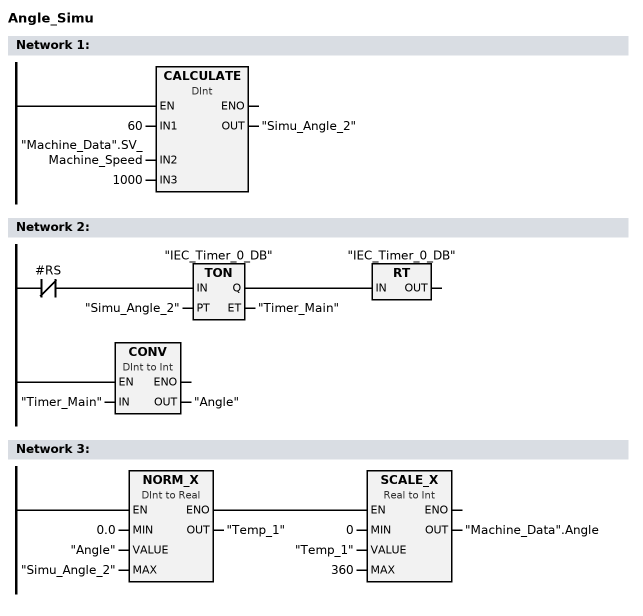
   RUNG wire#powerrail
      { S7_Templates := "SrcType := DInt"; S7_Expression := "IN1/IN2*IN3" } Calculate(in1 := 60, in2 := "Machine_Data".SV_Machine_Speed, in3 := 1000, out => "Simu_Angle_2")
   END_RUNG
   // the same network as SCL:
   "Simu_Angle_2" := 60/"Machine_Data".SV_Machine_Speed*1000;
END_REGION

REGION Network 2
   "IEC_Timer_0_DB".TON(IN := NOT #RS, PT := "Simu_Angle_2", ET => "Timer_Main");
   IF "IEC_Timer_0_DB".Q THEN RESET_TIMER("IEC_Timer_0_DB"); END_IF;
   "Angle" := DINT_TO_INT("Timer_Main");
END_REGION

REGION Network 3
   RUNG wire#powerrail
      { S7_Templates := "[SrcType := DInt, DestType := Real]" } Normalize(min := 0.0, value := "Angle", max := "Simu_Angle_2", out => "Temp_1")
      { S7_Templates := "[SrcType := Real, DestType := Int]" } Scale(min := 0, value := "Temp_1", max := 360, out => "Machine_Data".Angle)
   END_RUNG
   // the same network as SCL:
   "Temp_1" := NORM_X(MIN := 0.0, VALUE := "Angle", MAX := "Simu_Angle_2");
   "Machine_Data".Angle := SCALE_X(MIN := 0, VALUE := "Temp_1", MAX := 360);
END_REGION
END_FUNCTION

FUNCTION "Control_Via_Angle" : Void   // FC7, LAD
{ S7_Optimized_Access := 'TRUE' }
VERSION : 0.1
   VAR_INPUT
      Begin_Angle : Int;
      End_Angle : Int;
      Inter_Lock : Bool;
   END_VAR
   VAR_OUTPUT
      Set : Bool;
   END_VAR
   VAR_IN_OUT
      Enable : Bool;
   END_VAR
BEGIN

REGION Network 1
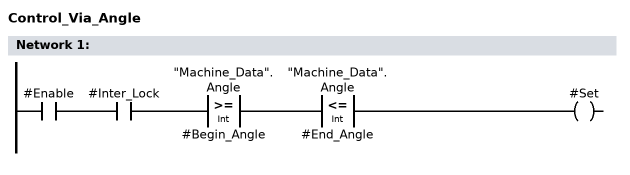
   RUNG wire#powerrail
      Contact( #Enable )
      Contact( #Inter_Lock )
      { S7_Templates := "SrcType := Int" } GE_Contact(in1 := "Machine_Data".Angle, in2 := #Begin_Angle)
      { S7_Templates := "SrcType := Int" } LE_Contact(in1 := "Machine_Data".Angle, in2 := #End_Angle)
      Coil( #Set )
   END_RUNG
   // the same network as SCL:
   #Set := #Enable AND #Inter_Lock AND ("Machine_Data".Angle >= #Begin_Angle) AND ("Machine_Data".Angle <= #End_Angle);
END_REGION
END_FUNCTION

FUNCTION "Servo_Pull" : Void   // FC8, LAD
{ S7_Optimized_Access := 'TRUE' }
VERSION : 0.1
BEGIN

REGION Network 1: CW
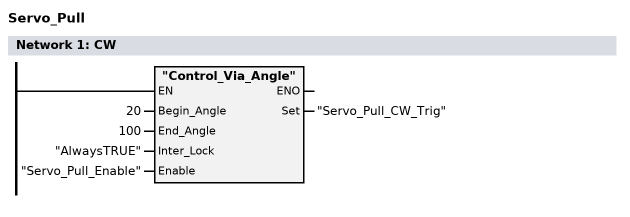
   RUNG wire#powerrail
      "Control_Via_Angle"(Begin_Angle := 20, End_Angle := 100, Inter_Lock := "AlwaysTRUE", Enable := "Servo_Pull_Enable", Set => "Servo_Pull_CW_Trig")
   END_RUNG
   // the same network as SCL:
   "Control_Via_Angle"(Begin_Angle := 20,
                       End_Angle := 100,
                       Inter_Lock := "AlwaysTRUE",
                       Enable := "Servo_Pull_Enable",
                       Set => "Servo_Pull_CW_Trig");
END_REGION
END_FUNCTION

FUNCTION "PinHole" : Void   // FC9, LAD
{ S7_Optimized_Access := 'TRUE' }
VERSION : 0.1
   VAR_TEMP   // added for the SCL form of the ladder/FBD networks
      _w1 : Bool;
      _w2 : Bool;
   END_VAR
BEGIN

REGION Network 1
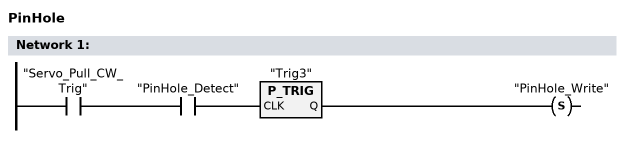
   RUNG wire#powerrail
      Contact( "Servo_Pull_CW_Trig" )
      Contact( "PinHole_Detect" )
      P_Trig( "Trig3" )
      S_Coil( "PinHole_Write" )
   END_RUNG
   // the same network as SCL:
   #_w1 := "Servo_Pull_CW_Trig" AND "PinHole_Detect";
   #_w2 := #_w1 AND NOT "Trig3";   // rising edge
   "Trig3" := #_w1;
   IF #_w2 THEN "PinHole_Write" := TRUE; END_IF;
END_REGION

REGION Network 2 (SCL)
   IF "PinHole_Write" = TRUE THEN
       "Blister_Animation".Blister_1["Station_Position".Cut_to_PinHole] := 2#000000;
       "Blister_Animation".Blister_Matrix["Station_Position".Cut_to_PinHole] := 2#000000;
       "PinHole_Write" := FALSE;

   END_IF;
END_REGION
END_FUNCTION

ORGANIZATION_BLOCK "Main"   // OB1, LAD, ProgramCycle
TITLE = "Main Program Sweep (Cycle)"
{ S7_Optimized_Access := 'TRUE' }
VERSION : 0.1
   VAR_INPUT
      Initial_Call : Bool;   // Initial call of this OB
      Remanence : Bool;   // =True, if remanent data are available
   END_VAR
   VAR_TEMP
      Trig_1 : Bool;
   END_VAR
   VAR_TEMP   // added for the SCL form of the ladder/FBD networks
      _w1 : Bool;
      _w2 : Bool;
   END_VAR
BEGIN

REGION Network 1: Conveyor
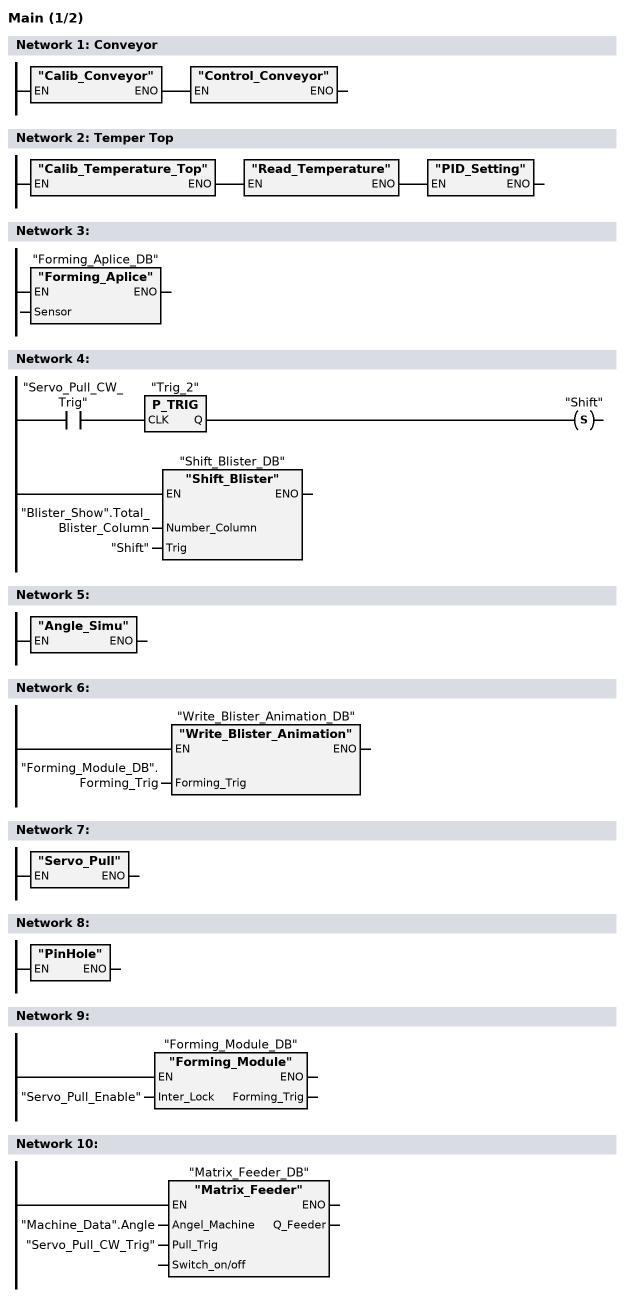
   RUNG wire#powerrail
      "Calib_Conveyor"()
      "Control_Conveyor"()
   END_RUNG
   // the same network as SCL:
   "Calib_Conveyor"(ENO => #_w1);
   IF #_w1 THEN "Control_Conveyor"(); END_IF;
END_REGION

REGION Network 2: Temper Top
   RUNG wire#powerrail
      "Calib_Temperature_Top"()
      "Read_Temperature"()
      "PID_Setting"()
   END_RUNG
   // the same network as SCL:
   "Calib_Temperature_Top"(ENO => #_w1);
   "Read_Temperature"(EN := #_w1, ENO => #_w2);
   IF #_w2 THEN "PID_Setting"(); END_IF;
END_REGION

REGION Network 3
   RUNG wire#powerrail
      "Forming_Aplice_DB"(Sensor :=)
   END_RUNG
   // the same network as SCL:
   "Forming_Aplice_DB"();   // "Forming_Aplice"
END_REGION

REGION Network 4
   RUNG wire#powerrail
      Contact( "Servo_Pull_CW_Trig" )
      P_Trig( "Trig_2" )
      S_Coil( "Shift" )
   END_RUNG
   RUNG wire#powerrail
      "Shift_Blister_DB"(Number_Column := "Blister_Show".Total_Blister_Column, Trig := "Shift")
   END_RUNG
   // the same network as SCL:
   #_w1 := "Servo_Pull_CW_Trig" AND NOT "Trig_2";   // rising edge
   "Trig_2" := "Servo_Pull_CW_Trig";
   IF #_w1 THEN "Shift" := TRUE; END_IF;
   "Shift_Blister_DB"(Number_Column := "Blister_Show".Total_Blister_Column, Trig := "Shift");   // "Shift_Blister"
END_REGION

REGION Network 5
   RUNG wire#powerrail
      "Angle_Simu"()
   END_RUNG
   // the same network as SCL:
   "Angle_Simu"();
END_REGION

REGION Network 6
   RUNG wire#powerrail
      "Write_Blister_Animation_DB"(Forming_Trig := "Forming_Module_DB".Forming_Trig)
   END_RUNG
   // the same network as SCL:
   "Write_Blister_Animation_DB"(Forming_Trig := "Forming_Module_DB".Forming_Trig);   // "Write_Blister_Animation"
END_REGION

REGION Network 7
   RUNG wire#powerrail
      "Servo_Pull"()
   END_RUNG
   // the same network as SCL:
   "Servo_Pull"();
END_REGION

REGION Network 8
   RUNG wire#powerrail
      "PinHole"()
   END_RUNG
   // the same network as SCL:
   "PinHole"();
END_REGION

REGION Network 9
   RUNG wire#powerrail
      "Forming_Module_DB"(Inter_Lock := "Servo_Pull_Enable", Forming_Trig =>)
   END_RUNG
   // the same network as SCL:
   "Forming_Module_DB"(Inter_Lock := "Servo_Pull_Enable");   // "Forming_Module"
END_REGION

REGION Network 10
   RUNG wire#powerrail
      "Matrix_Feeder_DB"(Angel_Machine := "Machine_Data".Angle, Pull_Trig := "Servo_Pull_CW_Trig", "Switch_on/off" :=, Q_Feeder =>)
   END_RUNG
   // the same network as SCL:
   "Matrix_Feeder_DB"(Angel_Machine := "Machine_Data".Angle, Pull_Trig := "Servo_Pull_CW_Trig");   // "Matrix_Feeder"
END_REGION

REGION Network 12
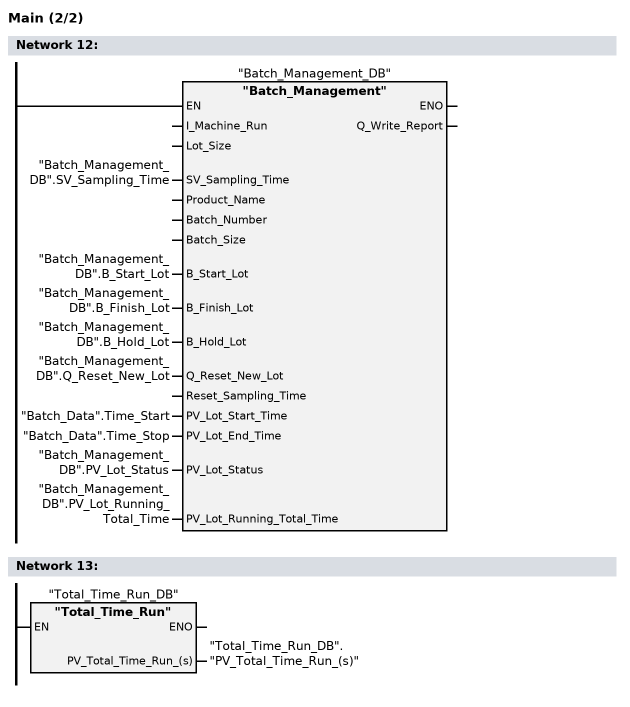
   RUNG wire#powerrail
      "Batch_Management_DB"(I_Machine_Run :=, Lot_Size :=, SV_Sampling_Time := "Batch_Management_DB".SV_Sampling_Time, Product_Name :=, Batch_Number :=, Batch_Size :=, B_Start_Lot := "Batch_Management_DB".B_Start_Lot, B_Finish_Lot := "Batch_Management_DB".B_Finish_Lot, B_Hold_Lot := "Batch_Management_DB".B_Hold_Lot, Q_Reset_New_Lot := "Batch_Management_DB".Q_Reset_New_Lot, Reset_Sampling_Time :=, PV_Lot_Start_Time := "Batch_Data".Time_Start, PV_Lot_End_Time := "Batch_Data".Time_Stop, PV_Lot_Status := "Batch_Management_DB".PV_Lot_Status, PV_Lot_Running_Total_Time := "Batch_Management_DB".PV_Lot_Running_Total_Time, Q_Write_Report =>)
   END_RUNG
   // the same network as SCL:
   "Batch_Management_DB"(SV_Sampling_Time := "Batch_Management_DB".SV_Sampling_Time,   // "Batch_Management"
                         B_Start_Lot := "Batch_Management_DB".B_Start_Lot,
                         B_Finish_Lot := "Batch_Management_DB".B_Finish_Lot,
                         B_Hold_Lot := "Batch_Management_DB".B_Hold_Lot,
                         Q_Reset_New_Lot := "Batch_Management_DB".Q_Reset_New_Lot,
                         PV_Lot_Start_Time := "Batch_Data".Time_Start,
                         PV_Lot_End_Time := "Batch_Data".Time_Stop,
                         PV_Lot_Status := "Batch_Management_DB".PV_Lot_Status,
                         PV_Lot_Running_Total_Time := "Batch_Management_DB".PV_Lot_Running_Total_Time);
END_REGION

REGION Network 13
   RUNG wire#powerrail
      "Total_Time_Run_DB"("PV_Total_Time_Run_(s)" => "Total_Time_Run_DB"."PV_Total_Time_Run_(s)")
   END_RUNG
   // the same network as SCL:
   "Total_Time_Run_DB"("PV_Total_Time_Run_(s)" => "Total_Time_Run_DB"."PV_Total_Time_Run_(s)");   // "Total_Time_Run"
END_REGION
END_ORGANIZATION_BLOCK

ORGANIZATION_BLOCK "Startup"   // OB100, LAD, Startup
TITLE = "Complete Restart"
{ S7_Optimized_Access := 'TRUE' }
VERSION : 0.1
   VAR_INPUT
      LostRetentive : Bool;   // True if retentive data are lost
      LostRTC : Bool;   // True if date and time are lost
   END_VAR
BEGIN
END_ORGANIZATION_BLOCK

// folder: FB_Calib

FUNCTION_BLOCK "Calib_Speed_Output"   // FB1, LAD
{ S7_Optimized_Access := 'TRUE' }
VERSION : 0.1
   VAR_INPUT
      Enable_Calib : Bool;
      Point_1_Analog_L : Int;
      Point_2_Analog_H : Int;
      Default_Analog_Min : Int;
      Default_Analog_Max : Int;
      Default_Speed_Min : Int;
      Default_Speed_Max : Int;
   END_VAR
   VAR_OUTPUT
      Result_Min_Analog : Int;
      Result_Max_Analog : Int;
      Result_Min_Speed : Int;
      Result_Max_Speed : Int;
      O_Analog : Int;
      O_Run : Bool;
      O_Result : Bool;
   END_VAR
   VAR_IN_OUT
      Dim_Point_1_Button : Bool;
      Dim_Point_2_Button : Bool;
      OK_Button : Bool;
      SV_Point_1_Speed : Int;
      SV_Point_2_Speed : Int;
      B_Default : Bool;
      B_Run_Min_Speed : Bool;
      B_Run_Max_Speed : Bool;
   END_VAR
   VAR
      Temp_Value : Real;
      Temp_1 : Int;
      Temp_2 : Int;
      Temp_3 : Int;
      Temp_4 : Int;
      Trig1 : Bool;
      Trig2 : Bool;
      T1 : IEC_TIMER;
      T2 : IEC_TIMER;
      T3 : IEC_TIMER;
   END_VAR
   VAR_TEMP   // added for the SCL form of the ladder/FBD networks
      _w1 : Bool;
      _w2 : Bool;
      _w3 : Bool;
      _w4 : Bool;
      _w5 : Bool;
   END_VAR
BEGIN

REGION Network 1: Run speed min max
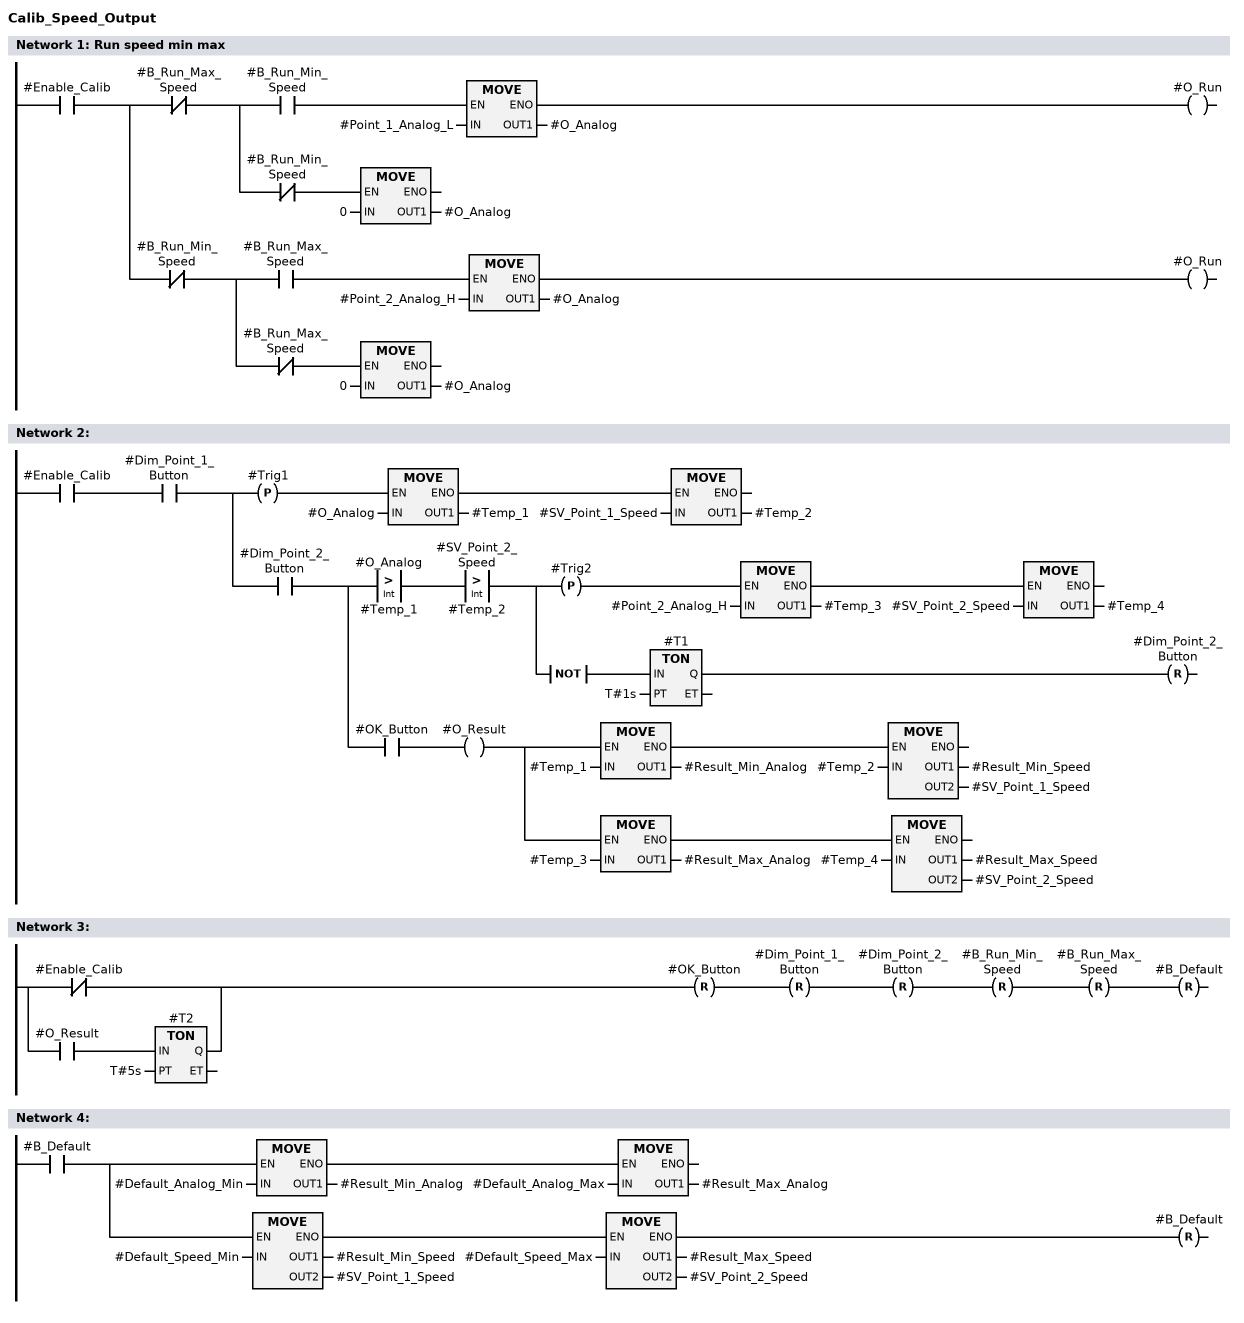
   RUNG wire#powerrail
      Contact( #Enable_Calib )
      wire#w1
      I_Contact( #B_Run_Max_Speed )
      wire#w2
      Contact( #B_Run_Min_Speed )
      Move(in := #Point_1_Analog_L, out1 => #O_Analog)
      Coil( #O_Run )
   END_RUNG
   RUNG wire#w2
      I_Contact( #B_Run_Min_Speed )
      Move(in := 0, out1 => #O_Analog)
   END_RUNG
   RUNG wire#w1
      I_Contact( #B_Run_Min_Speed )
      wire#w3
      Contact( #B_Run_Max_Speed )
      Move(in := #Point_2_Analog_H, out1 => #O_Analog)
      Coil( #O_Run )
   END_RUNG
   RUNG wire#w3
      I_Contact( #B_Run_Max_Speed )
      Move(in := 0, out1 => #O_Analog)
   END_RUNG
   // the same network as SCL:
   #_w1 := #Enable_Calib AND NOT #B_Run_Max_Speed;
   #_w2 := #_w1 AND #B_Run_Min_Speed;
   IF #_w2 THEN #O_Analog := #Point_1_Analog_L; END_IF;
   #O_Run := #_w2;
   IF #_w1 AND NOT #B_Run_Min_Speed THEN #O_Analog := 0; END_IF;
   #_w3 := #Enable_Calib AND NOT #B_Run_Min_Speed;
   #_w4 := #_w3 AND #B_Run_Max_Speed;
   IF #_w4 THEN #O_Analog := #Point_2_Analog_H; END_IF;
   #O_Run := #_w4;
   IF #_w3 AND NOT #B_Run_Max_Speed THEN #O_Analog := 0; END_IF;
END_REGION

REGION Network 2
   #_w1 := #Enable_Calib AND #Dim_Point_1_Button;
   #_w2 := #_w1 AND NOT #Trig1;   // rising edge
   #Trig1 := #_w1;
   IF #_w2 THEN
       #Temp_1 := #O_Analog;
       #Temp_2 := #SV_Point_1_Speed;
   END_IF;
   #_w3 := #_w1 AND #Dim_Point_2_Button;
   #_w4 := #_w3 AND (#O_Analog > #Temp_1) AND (#SV_Point_2_Speed > #Temp_2);
   #_w5 := #_w4 AND NOT #Trig2;   // rising edge
   #Trig2 := #_w4;
   IF #_w5 THEN
       #Temp_3 := #Point_2_Analog_H;
       #Temp_4 := #SV_Point_2_Speed;
   END_IF;
   #T1.TON(IN := NOT #_w4, PT := T#1s);
   IF #T1.Q THEN #Dim_Point_2_Button := FALSE; END_IF;
   #O_Result := #_w3 AND #OK_Button;
   IF #O_Result THEN
       #Result_Min_Analog := #Temp_1;
       #Result_Min_Speed := #Temp_2;
       #SV_Point_1_Speed := #Temp_2;
       #Result_Max_Analog := #Temp_3;
       #Result_Max_Speed := #Temp_4;
       #SV_Point_2_Speed := #Temp_4;
   END_IF;
END_REGION

REGION Network 3
   #T2.TON(IN := #O_Result, PT := T#5s);
   IF NOT #Enable_Calib OR #T2.Q THEN
       #OK_Button := FALSE;
       #Dim_Point_1_Button := FALSE;
       #Dim_Point_2_Button := FALSE;
       #B_Run_Min_Speed := FALSE;
       #B_Run_Max_Speed := FALSE;
       #B_Default := FALSE;
   END_IF;
END_REGION

REGION Network 4
   RUNG wire#powerrail
      Contact( #B_Default )
      wire#w1
      Move(in := #Default_Analog_Min, out1 => #Result_Min_Analog)
      Move(in := #Default_Analog_Max, out1 => #Result_Max_Analog)
   END_RUNG
   RUNG wire#w1
      Move(in := #Default_Speed_Min, out1 => #Result_Min_Speed, out2 => #SV_Point_1_Speed)
      Move(in := #Default_Speed_Max, out1 => #Result_Max_Speed, out2 => #SV_Point_2_Speed)
      R_Coil( #B_Default )
   END_RUNG
   // the same network as SCL:
   IF #B_Default THEN
       #Result_Min_Analog := #Default_Analog_Min;
       #Result_Max_Analog := #Default_Analog_Max;
       #Result_Min_Speed := #Default_Speed_Min;
       #SV_Point_1_Speed := #Default_Speed_Min;
       #Result_Max_Speed := #Default_Speed_Max;
       #SV_Point_2_Speed := #Default_Speed_Max;
       #B_Default := FALSE;
   END_IF;
END_REGION
END_FUNCTION_BLOCK

FUNCTION_BLOCK "Calib_Temperature_Input"   // FB3, LAD
{ S7_Optimized_Access := 'TRUE' }
VERSION : 0.1
   VAR_INPUT
      Enable_Calib : Bool;
      I_Analog_Read : Int;
      Default_Analog_Min : Int;
      Default_Analog_Max : Int;
      Default_Temper_Min : Int;
      Default_Temper_Max : Int;
   END_VAR
   VAR_OUTPUT
      Min_Analog : Int;
      Max_Analog : Int;
      Min_Temper : Int;
      Max_Temper : Int;
      Result_Calib : Bool;
   END_VAR
   VAR_IN_OUT
      Dim_Point_1_Button : Bool;
      Dim_Point_2_Button : Bool;
      OK_Button : Bool;
      Default_Button : Bool;
      SV_Temper_1 : Int;
      SV_Temper_2 : Int;
   END_VAR
   VAR
      Temp_Value : Real;
      Temp_1 : Int;
      Temp_2 : Int;
      Temp_3 : Int;
      Temp_4 : Int;
      Button_2_Pressed : Bool;
      Trig_1 : Bool;
      Timer_1 : IEC_TIMER;
      Timer_2 : IEC_TIMER;
      Timer_3 : IEC_TIMER;
      Point_1_Sucess : Bool;
      Point_2_Sucess : Bool;
      Timer_4 : IEC_TIMER;
      Trig_2 : Bool;
      Trig_3 : Bool;
   END_VAR
   VAR_TEMP   // added for the SCL form of the ladder/FBD networks
      _w1 : Bool;
      _w2 : Bool;
      _w3 : Bool;
      _w4 : Bool;
   END_VAR
BEGIN

REGION Network 1
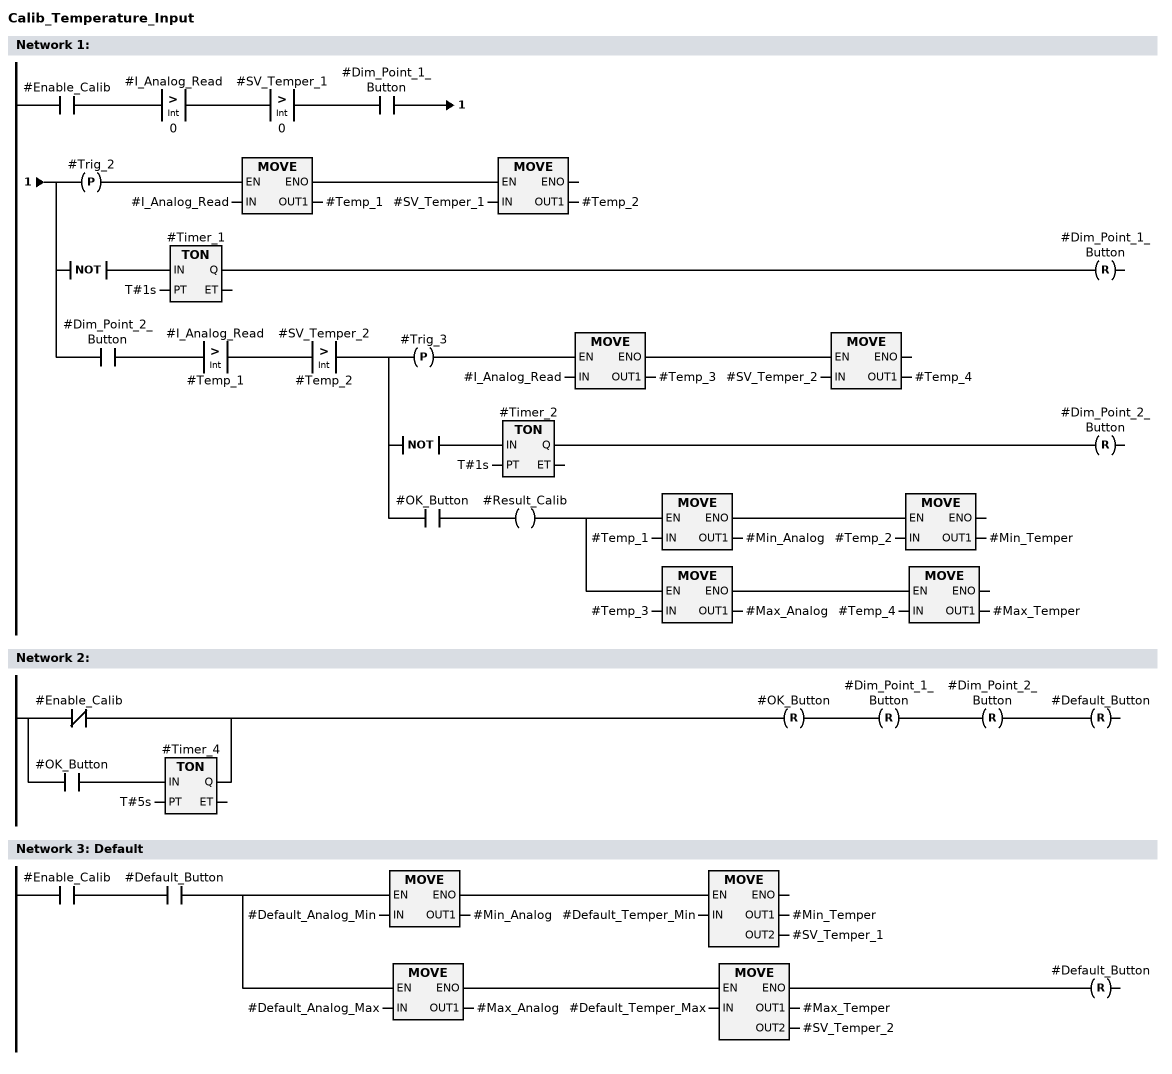
   #_w1 := #Enable_Calib AND (#I_Analog_Read > 0) AND (#SV_Temper_1 > 0) AND #Dim_Point_1_Button;
   #_w2 := #_w1 AND NOT #Trig_2;   // rising edge
   #Trig_2 := #_w1;
   IF #_w2 THEN
       #Temp_1 := #I_Analog_Read;
       #Temp_2 := #SV_Temper_1;
   END_IF;
   #Timer_1.TON(IN := NOT #_w1, PT := T#1s);
   IF #Timer_1.Q THEN #Dim_Point_1_Button := FALSE; END_IF;
   #_w3 := #_w1 AND #Dim_Point_2_Button AND (#I_Analog_Read > #Temp_1) AND (#SV_Temper_2 > #Temp_2);
   #_w4 := #_w3 AND NOT #Trig_3;   // rising edge
   #Trig_3 := #_w3;
   IF #_w4 THEN
       #Temp_3 := #I_Analog_Read;
       #Temp_4 := #SV_Temper_2;
   END_IF;
   #Timer_2.TON(IN := NOT #_w3, PT := T#1s);
   IF #Timer_2.Q THEN #Dim_Point_2_Button := FALSE; END_IF;
   #Result_Calib := #_w3 AND #OK_Button;
   IF #Result_Calib THEN
       #Min_Analog := #Temp_1;
       #Min_Temper := #Temp_2;
       #Max_Analog := #Temp_3;
       #Max_Temper := #Temp_4;
   END_IF;
END_REGION

REGION Network 2
   #Timer_4.TON(IN := #OK_Button, PT := T#5s);
   IF NOT #Enable_Calib OR #Timer_4.Q THEN
       #OK_Button := FALSE;
       #Dim_Point_1_Button := FALSE;
       #Dim_Point_2_Button := FALSE;
       #Default_Button := FALSE;
   END_IF;
END_REGION

REGION Network 3: Default
   RUNG wire#powerrail
      Contact( #Enable_Calib )
      Contact( #Default_Button )
      wire#w1
      Move(in := #Default_Analog_Min, out1 => #Min_Analog)
      Move(in := #Default_Temper_Min, out1 => #Min_Temper, out2 => #SV_Temper_1)
   END_RUNG
   RUNG wire#w1
      Move(in := #Default_Analog_Max, out1 => #Max_Analog)
      Move(in := #Default_Temper_Max, out1 => #Max_Temper, out2 => #SV_Temper_2)
      R_Coil( #Default_Button )
   END_RUNG
   // the same network as SCL:
   IF #Enable_Calib AND #Default_Button THEN
       #Min_Analog := #Default_Analog_Min;
       #Min_Temper := #Default_Temper_Min;
       #SV_Temper_1 := #Default_Temper_Min;
       #Max_Analog := #Default_Analog_Max;
       #Max_Temper := #Default_Temper_Max;
       #SV_Temper_2 := #Default_Temper_Max;
       #Default_Button := FALSE;
   END_IF;
END_REGION
END_FUNCTION_BLOCK

// folder: FB_Scale

FUNCTION_BLOCK "Scale_Analog_Output"   // FB2, LAD
{ S7_Optimized_Access := 'TRUE' }
VERSION : 0.1
   VAR_INPUT
      Value_Norm : Real;
      Min_Norm : Real;
      Max_Norm : Real;
      Min_Scale : Real;
      Max_Scale : Real;
   END_VAR
   VAR_OUTPUT
      Out_Scale : Int;
   END_VAR
   VAR
      Temp : Real;
      Temp_2 : Real;
   END_VAR
BEGIN

REGION Network 1
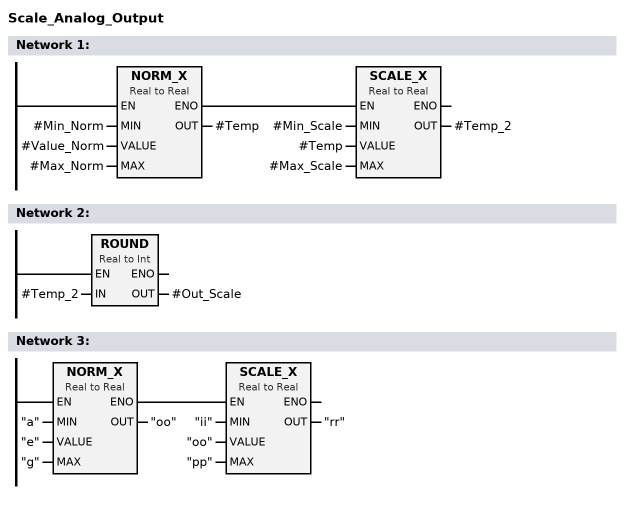
   RUNG wire#powerrail
      { S7_Templates := "[SrcType := Real, DestType := Real]" } Normalize(min := #Min_Norm, value := #Value_Norm, max := #Max_Norm, out => #Temp)
      { S7_Templates := "[SrcType := Real, DestType := Real]" } Scale(min := #Min_Scale, value := #Temp, max := #Max_Scale, out => #Temp_2)
   END_RUNG
   // the same network as SCL:
   #Temp := NORM_X(MIN := #Min_Norm, VALUE := #Value_Norm, MAX := #Max_Norm);
   #Temp_2 := SCALE_X(MIN := #Min_Scale, VALUE := #Temp, MAX := #Max_Scale);
END_REGION

REGION Network 2
   RUNG wire#powerrail
      { S7_Templates := "[SrcType := Real, DestType := Int]" } Round(in := #Temp_2, out => #Out_Scale)
   END_RUNG
   // the same network as SCL:
   #Out_Scale := ROUND(#Temp_2);
END_REGION

REGION Network 3
   RUNG wire#powerrail
      { S7_Templates := "[SrcType := Real, DestType := Real]" } Normalize(min := "a", value := "e", max := "g", out => "oo")
      { S7_Templates := "[SrcType := Real, DestType := Real]" } Scale(min := "ii", value := "oo", max := "pp", out => "rr")
   END_RUNG
   // the same network as SCL:
   "oo" := NORM_X(MIN := "a", VALUE := "e", MAX := "g");
   "rr" := SCALE_X(MIN := "ii", VALUE := "oo", MAX := "pp");
END_REGION
END_FUNCTION_BLOCK

FUNCTION_BLOCK "Scale_Analog_Input"   // FB4, LAD
{ S7_Optimized_Access := 'TRUE' }
VERSION : 0.1
   VAR_INPUT
      I_Analog : Int;
      Min_Analog : Int;
      Max_Analog : Int;
      Min_Temper : Int;
      Max_Temper : Int;
   END_VAR
   VAR_OUTPUT
      PV_Temp : Int;
   END_VAR
   VAR
      Temp : Real;
   END_VAR
BEGIN

REGION Network 1
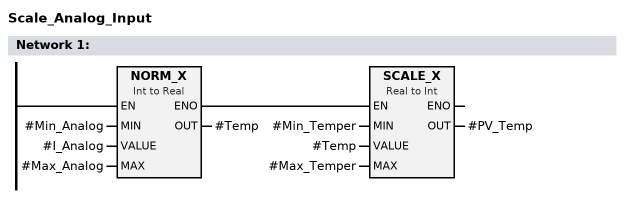
   RUNG wire#powerrail
      { S7_Templates := "[SrcType := Int, DestType := Real]" } Normalize(min := #Min_Analog, value := #I_Analog, max := #Max_Analog, out => #Temp)
      { S7_Templates := "[SrcType := Real, DestType := Int]" } Scale(min := #Min_Temper, value := #Temp, max := #Max_Temper, out => #PV_Temp)
   END_RUNG
   // the same network as SCL:
   #Temp := NORM_X(MIN := #Min_Analog, VALUE := #I_Analog, MAX := #Max_Analog);
   #PV_Temp := SCALE_X(MIN := #Min_Temper, VALUE := #Temp, MAX := #Max_Temper);
END_REGION
END_FUNCTION_BLOCK

// folder: Main_program/Conveyor

FUNCTION "Calib_Conveyor" : Void   // FC1, LAD
{ S7_Optimized_Access := 'TRUE' }
VERSION : 0.1
BEGIN

REGION Network 1: Xuat Analog
END_REGION

REGION Network 2
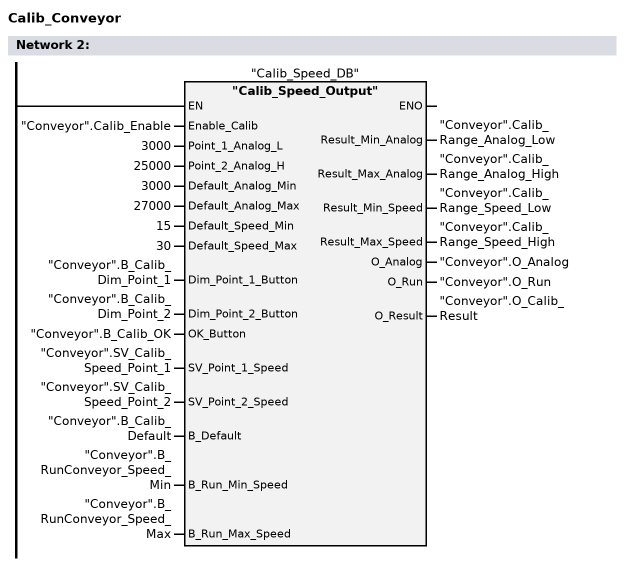
   RUNG wire#powerrail
      "Calib_Speed_DB"(Enable_Calib := "Conveyor".Calib_Enable, Point_1_Analog_L := 3000, Point_2_Analog_H := 25000, Default_Analog_Min := 3000, Default_Analog_Max := 27000, Default_Speed_Min := 15, Default_Speed_Max := 30, Dim_Point_1_Button := "Conveyor".B_Calib_Dim_Point_1, Dim_Point_2_Button := "Conveyor".B_Calib_Dim_Point_2, OK_Button := "Conveyor".B_Calib_OK, SV_Point_1_Speed := "Conveyor".SV_Calib_Speed_Point_1, SV_Point_2_Speed := "Conveyor".SV_Calib_Speed_Point_2, B_Default := "Conveyor".B_Calib_Default, B_Run_Min_Speed := "Conveyor".B_RunConveyor_Speed_Min, B_Run_Max_Speed := "Conveyor".B_RunConveyor_Speed_Max, Result_Min_Analog => "Conveyor".Calib_Range_Analog_Low, Result_Max_Analog => "Conveyor".Calib_Range_Analog_High, Result_Min_Speed => "Conveyor".Calib_Range_Speed_Low, Result_Max_Speed => "Conveyor".Calib_Range_Speed_High, O_Analog => "Conveyor".O_Analog, O_Run => "Conveyor".O_Run, O_Result => "Conveyor".O_Calib_Result)
   END_RUNG
   // the same network as SCL:
   "Calib_Speed_DB"(Enable_Calib := "Conveyor".Calib_Enable,   // "Calib_Speed_Output"
                    Point_1_Analog_L := 3000,
                    Point_2_Analog_H := 25000,
                    Default_Analog_Min := 3000,
                    Default_Analog_Max := 27000,
                    Default_Speed_Min := 15,
                    Default_Speed_Max := 30,
                    Dim_Point_1_Button := "Conveyor".B_Calib_Dim_Point_1,
                    Dim_Point_2_Button := "Conveyor".B_Calib_Dim_Point_2,
                    OK_Button := "Conveyor".B_Calib_OK,
                    SV_Point_1_Speed := "Conveyor".SV_Calib_Speed_Point_1,
                    SV_Point_2_Speed := "Conveyor".SV_Calib_Speed_Point_2,
                    B_Default := "Conveyor".B_Calib_Default,
                    B_Run_Min_Speed := "Conveyor".B_RunConveyor_Speed_Min,
                    B_Run_Max_Speed := "Conveyor".B_RunConveyor_Speed_Max,
                    Result_Min_Analog => "Conveyor".Calib_Range_Analog_Low,
                    Result_Max_Analog => "Conveyor".Calib_Range_Analog_High,
                    Result_Min_Speed => "Conveyor".Calib_Range_Speed_Low,
                    Result_Max_Speed => "Conveyor".Calib_Range_Speed_High,
                    O_Analog => "Conveyor".O_Analog,
                    O_Run => "Conveyor".O_Run,
                    O_Result => "Conveyor".O_Calib_Result);
END_REGION
END_FUNCTION

FUNCTION "Control_Conveyor" : Void   // FC2, LAD
{ S7_Optimized_Access := 'TRUE' }
VERSION : 0.1
BEGIN

REGION Network 1
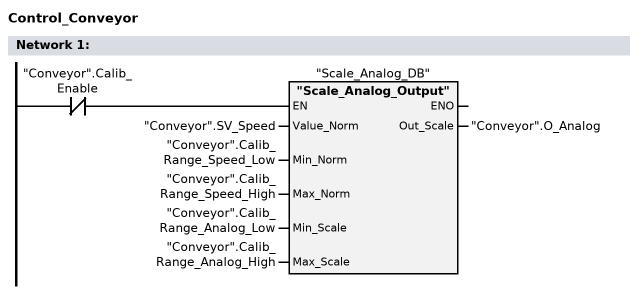
   RUNG wire#powerrail
      I_Contact( "Conveyor".Calib_Enable )
      "Scale_Analog_DB"(Value_Norm := "Conveyor".SV_Speed, Min_Norm := "Conveyor".Calib_Range_Speed_Low, Max_Norm := "Conveyor".Calib_Range_Speed_High, Min_Scale := "Conveyor".Calib_Range_Analog_Low, Max_Scale := "Conveyor".Calib_Range_Analog_High, Out_Scale => "Conveyor".O_Analog)
   END_RUNG
   // the same network as SCL:
   IF NOT "Conveyor".Calib_Enable THEN
       "Scale_Analog_DB"(Value_Norm := "Conveyor".SV_Speed,   // "Scale_Analog_Output"
                         Min_Norm := "Conveyor".Calib_Range_Speed_Low,
                         Max_Norm := "Conveyor".Calib_Range_Speed_High,
                         Min_Scale := "Conveyor".Calib_Range_Analog_Low,
                         Max_Scale := "Conveyor".Calib_Range_Analog_High,
                         Out_Scale => "Conveyor".O_Analog);
   END_IF;
END_REGION
END_FUNCTION

FUNCTION "PID_Setting" : Void   // FC5, LAD
{ S7_Optimized_Access := 'TRUE' }
VERSION : 0.1
BEGIN

REGION Network 1
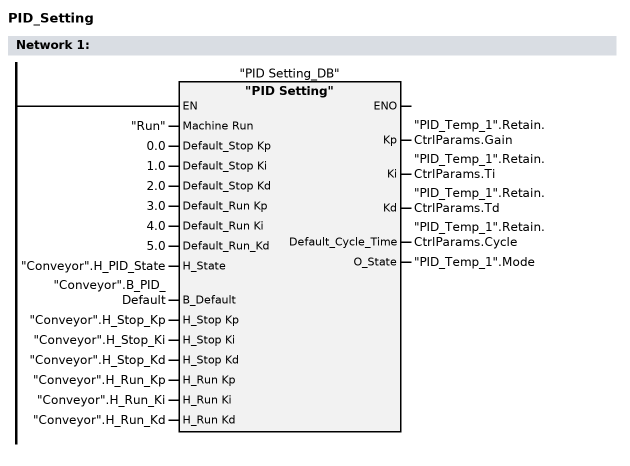
   RUNG wire#powerrail
      "PID Setting_DB"("Machine Run" := "Run", "Default_Stop Kp" := 0.0, "Default_Stop Ki" := 1.0, "Default_Stop Kd" := 2.0, "Default_Run Kp" := 3.0, "Default_Run Ki" := 4.0, Default_Run_Kd := 5.0, H_State := "Conveyor".H_PID_State, B_Default := "Conveyor".B_PID_Default, "H_Stop Kp" := "Conveyor".H_Stop_Kp, "H_Stop Ki" := "Conveyor".H_Stop_Ki, "H_Stop Kd" := "Conveyor".H_Stop_Kd, "H_Run Kp" := "Conveyor".H_Run_Kp, "H_Run Ki" := "Conveyor".H_Run_Ki, "H_Run Kd" := "Conveyor".H_Run_Kd, Kp => "PID_Temp_1".Retain.CtrlParams.Gain, Ki => "PID_Temp_1".Retain.CtrlParams.Ti, Kd => "PID_Temp_1".Retain.CtrlParams.Td, Default_Cycle_Time => "PID_Temp_1".Retain.CtrlParams.Cycle, O_State => "PID_Temp_1".Mode)
   END_RUNG
   // the same network as SCL:
   "PID Setting_DB"("Machine Run" := "Run",   // "PID Setting"
                    "Default_Stop Kp" := 0.0,
                    "Default_Stop Ki" := 1.0,
                    "Default_Stop Kd" := 2.0,
                    "Default_Run Kp" := 3.0,
                    "Default_Run Ki" := 4.0,
                    Default_Run_Kd := 5.0,
                    H_State := "Conveyor".H_PID_State,
                    B_Default := "Conveyor".B_PID_Default,
                    "H_Stop Kp" := "Conveyor".H_Stop_Kp,
                    "H_Stop Ki" := "Conveyor".H_Stop_Ki,
                    "H_Stop Kd" := "Conveyor".H_Stop_Kd,
                    "H_Run Kp" := "Conveyor".H_Run_Kp,
                    "H_Run Ki" := "Conveyor".H_Run_Ki,
                    "H_Run Kd" := "Conveyor".H_Run_Kd,
                    Kp => "PID_Temp_1".Retain.CtrlParams.Gain,
                    Ki => "PID_Temp_1".Retain.CtrlParams.Ti,
                    Kd => "PID_Temp_1".Retain.CtrlParams.Td,
                    Default_Cycle_Time => "PID_Temp_1".Retain.CtrlParams.Cycle,
                    O_State => "PID_Temp_1".Mode);
END_REGION
END_FUNCTION

// folder: Main_program/Temperature_Top

FUNCTION "Calib_Temperature_Top" : Void   // FC3, LAD
{ S7_Optimized_Access := 'TRUE' }
VERSION : 0.1
BEGIN

REGION Network 1
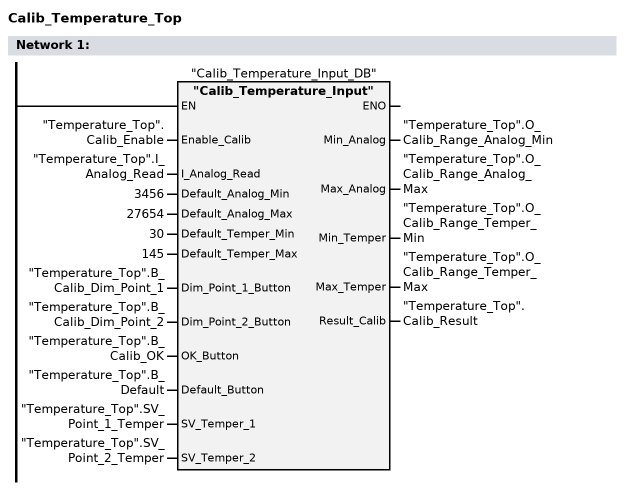
   RUNG wire#powerrail
      "Calib_Temperature_Input_DB"(Enable_Calib := "Temperature_Top".Calib_Enable, I_Analog_Read := "Temperature_Top".I_Analog_Read, Default_Analog_Min := 3456, Default_Analog_Max := 27654, Default_Temper_Min := 30, Default_Temper_Max := 145, Dim_Point_1_Button := "Temperature_Top".B_Calib_Dim_Point_1, Dim_Point_2_Button := "Temperature_Top".B_Calib_Dim_Point_2, OK_Button := "Temperature_Top".B_Calib_OK, Default_Button := "Temperature_Top".B_Default, SV_Temper_1 := "Temperature_Top".SV_Point_1_Temper, SV_Temper_2 := "Temperature_Top".SV_Point_2_Temper, Min_Analog => "Temperature_Top".O_Calib_Range_Analog_Min, Max_Analog => "Temperature_Top".O_Calib_Range_Analog_Max, Min_Temper => "Temperature_Top".O_Calib_Range_Temper_Min, Max_Temper => "Temperature_Top".O_Calib_Range_Temper_Max, Result_Calib => "Temperature_Top".Calib_Result)
   END_RUNG
   // the same network as SCL:
   "Calib_Temperature_Input_DB"(Enable_Calib := "Temperature_Top".Calib_Enable,   // "Calib_Temperature_Input"
                           I_Analog_Read := "Temperature_Top".I_Analog_Read,
                           Default_Analog_Min := 3456,
                           Default_Analog_Max := 27654,
                           Default_Temper_Min := 30,
                           Default_Temper_Max := 145,
                           Dim_Point_1_Button := "Temperature_Top".B_Calib_Dim_Point_1,
                           Dim_Point_2_Button := "Temperature_Top".B_Calib_Dim_Point_2,
                           OK_Button := "Temperature_Top".B_Calib_OK,
                           Default_Button := "Temperature_Top".B_Default,
                           SV_Temper_1 := "Temperature_Top".SV_Point_1_Temper,
                           SV_Temper_2 := "Temperature_Top".SV_Point_2_Temper,
                           Min_Analog => "Temperature_Top".O_Calib_Range_Analog_Min,
                           Max_Analog => "Temperature_Top".O_Calib_Range_Analog_Max,
                           Min_Temper => "Temperature_Top".O_Calib_Range_Temper_Min,
                           Max_Temper => "Temperature_Top".O_Calib_Range_Temper_Max,
                           Result_Calib => "Temperature_Top".Calib_Result);
END_REGION
END_FUNCTION

FUNCTION "Read_Temperature" : Void   // FC4, LAD
{ S7_Optimized_Access := 'TRUE' }
VERSION : 0.1
   VAR_TEMP
      Err : DWord;
      Trig_1 : Bool;
      OH : Real;
      OC : Real;
      OHP : Int;
      OCP : Int;
   END_VAR
   VAR_TEMP   // added for the SCL form of the ladder/FBD networks
      _w1 : Bool;
      _w2 : Bool;
   END_VAR
BEGIN

REGION Network 1
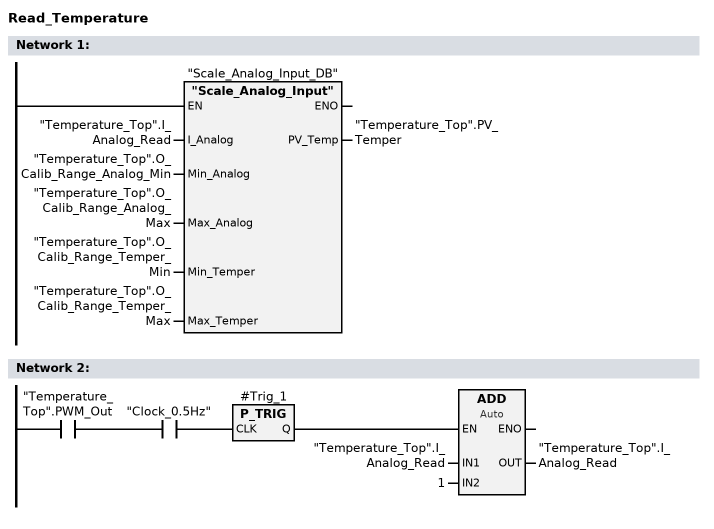
   RUNG wire#powerrail
      "Scale_Analog_Input_DB"(I_Analog := "Temperature_Top".I_Analog_Read, Min_Analog := "Temperature_Top".O_Calib_Range_Analog_Min, Max_Analog := "Temperature_Top".O_Calib_Range_Analog_Max, Min_Temper := "Temperature_Top".O_Calib_Range_Temper_Min, Max_Temper := "Temperature_Top".O_Calib_Range_Temper_Max, PV_Temp => "Temperature_Top".PV_Temper)
   END_RUNG
   // the same network as SCL:
   "Scale_Analog_Input_DB"(I_Analog := "Temperature_Top".I_Analog_Read,   // "Scale_Analog_Input"
                           Min_Analog := "Temperature_Top".O_Calib_Range_Analog_Min,
                           Max_Analog := "Temperature_Top".O_Calib_Range_Analog_Max,
                           Min_Temper := "Temperature_Top".O_Calib_Range_Temper_Min,
                           Max_Temper := "Temperature_Top".O_Calib_Range_Temper_Max,
                           PV_Temp => "Temperature_Top".PV_Temper);
END_REGION

REGION Network 2
   RUNG wire#powerrail
      Contact( "Temperature_Top".PWM_Out )
      Contact( "Clock_0.5Hz" )
      P_Trig( #Trig_1 )
      Add(in1 := "Temperature_Top".I_Analog_Read, in2 := 1, out => "Temperature_Top".I_Analog_Read)
   END_RUNG
   // the same network as SCL:
   #_w1 := "Temperature_Top".PWM_Out AND "Clock_0.5Hz";
   #_w2 := #_w1 AND NOT #Trig_1;   // rising edge
   #Trig_1 := #_w1;
   IF #_w2 THEN "Temperature_Top".I_Analog_Read := "Temperature_Top".I_Analog_Read + 1; END_IF;
END_REGION
END_FUNCTION

// folder: PID_Setting

FUNCTION_BLOCK "PID Setting"   // FB5, LAD
{ S7_Optimized_Access := 'TRUE' }
VERSION : 0.1
   VAR_INPUT
      "Machine Run" : Bool;
      "Default_Stop Kp" : Real;
      "Default_Stop Ki" : Real;
      "Default_Stop Kd" : Real;
      "Default_Run Kp" : Real;
      "Default_Run Ki" : Real;
      Default_Run_Kd : Real;
   END_VAR
   VAR_OUTPUT
      Kp : Real;
      Ki : Real;
      Kd : Real;
      Default_Cycle_Time : Real;
      O_State : Int;
   END_VAR
   VAR_IN_OUT
      H_State : Int := 3;
      B_Default : Bool;
      "H_Stop Kp" : Real;
      "H_Stop Ki" : Real;
      "H_Stop Kd" : Real;
      "H_Run Kp" : Real;
      "H_Run Ki" : Real;
      "H_Run Kd" : Real;
   END_VAR
   VAR
      T : IEC_TIMER;
   END_VAR
BEGIN

REGION Network 1: Default
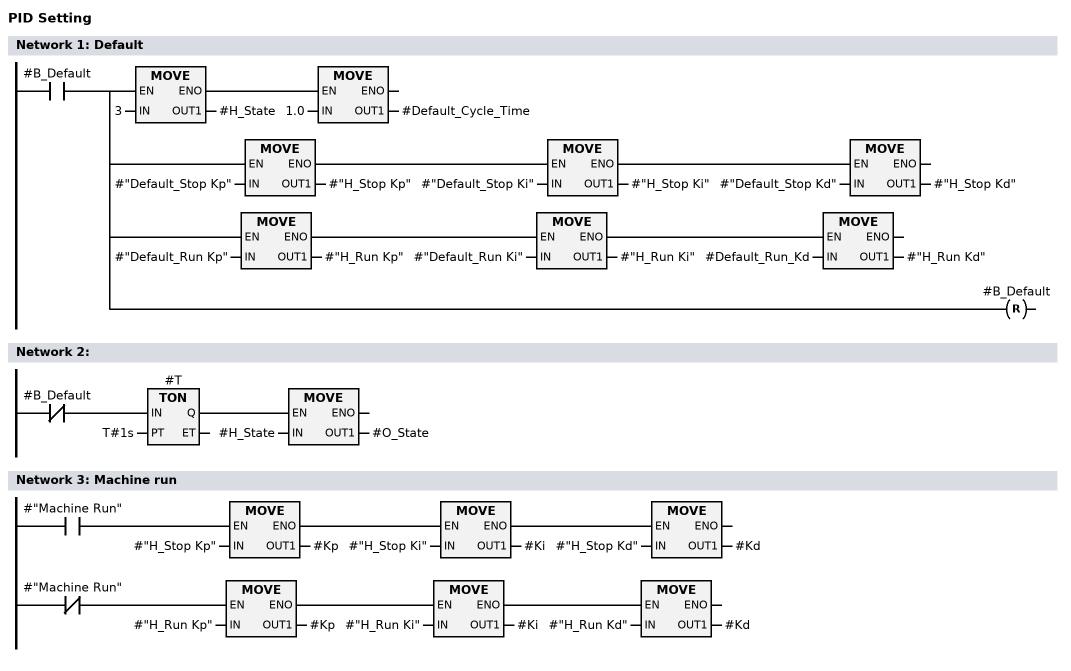
   RUNG wire#powerrail
      Contact( #B_Default )
      wire#w1
      Move(in := 3, out1 => #H_State)
      Move(in := 1.0, out1 => #Default_Cycle_Time)
   END_RUNG
   RUNG wire#w1
      Move(in := #"Default_Stop Kp", out1 => #"H_Stop Kp")
      Move(in := #"Default_Stop Ki", out1 => #"H_Stop Ki")
      Move(in := #"Default_Stop Kd", out1 => #"H_Stop Kd")
   END_RUNG
   RUNG wire#w1
      Move(in := #"Default_Run Kp", out1 => #"H_Run Kp")
      Move(in := #"Default_Run Ki", out1 => #"H_Run Ki")
      Move(in := #Default_Run_Kd, out1 => #"H_Run Kd")
   END_RUNG
   RUNG wire#w1
      R_Coil( #B_Default )
   END_RUNG
   // the same network as SCL:
   IF #B_Default THEN
       #H_State := 3;
       #Default_Cycle_Time := 1.0;
       #"H_Stop Kp" := #"Default_Stop Kp";
       #"H_Stop Ki" := #"Default_Stop Ki";
       #"H_Stop Kd" := #"Default_Stop Kd";
       #"H_Run Kp" := #"Default_Run Kp";
       #"H_Run Ki" := #"Default_Run Ki";
       #"H_Run Kd" := #Default_Run_Kd;
       #B_Default := FALSE;
   END_IF;
END_REGION

REGION Network 2
   #T.TON(IN := NOT #B_Default, PT := T#1s);
   IF #T.Q THEN #O_State := #H_State; END_IF;
END_REGION

REGION Network 3: Machine run
   RUNG wire#powerrail
      Contact( #"Machine Run" )
      Move(in := #"H_Stop Kp", out1 => #Kp)
      Move(in := #"H_Stop Ki", out1 => #Ki)
      Move(in := #"H_Stop Kd", out1 => #Kd)
   END_RUNG
   RUNG wire#powerrail
      I_Contact( #"Machine Run" )
      Move(in := #"H_Run Kp", out1 => #Kp)
      Move(in := #"H_Run Ki", out1 => #Ki)
      Move(in := #"H_Run Kd", out1 => #Kd)
   END_RUNG
   // the same network as SCL:
   IF #"Machine Run" THEN
       #Kp := #"H_Stop Kp";
       #Ki := #"H_Stop Ki";
       #Kd := #"H_Stop Kd";
   END_IF;
   IF NOT #"Machine Run" THEN
       #Kp := #"H_Run Kp";
       #Ki := #"H_Run Ki";
       #Kd := #"H_Run Kd";
   END_IF;
END_REGION
END_FUNCTION_BLOCK

(* ===== HMI "HMI_RT_1" =====
system functions are stored by id; their names below are inferred from use
connection "HMI_Connection_1": ETHERNET, S7_1200_OMS

HMI tags "Default tag table"
   "Conveyor_Calib_Enable" : Bool = PLC Conveyor.Calib_Enable, 100 ms
   "Conveyor_Calib_Dim_Point_1" : Bool = PLC Conveyor.B_Calib_Dim_Point_1, 100 ms
   "Conveyor_Calib_Dim_Point_2" : Bool = PLC Conveyor.B_Calib_Dim_Point_2, 100 ms
   "Conveyor_Calib_Speed_1" : Int = PLC Conveyor.SV_Calib_Speed_Point_1, 100 ms
   "Conveyor_Calib_Speed_2" : Int = PLC Conveyor.SV_Calib_Speed_Point_2, 100 ms
   "Conveyor_B_RunConveyor_Speed_Min" : Bool = PLC Conveyor.B_RunConveyor_Speed_Min, 100 ms
   "Conveyor_B_RunConveyor_Speed_Max" : Bool = PLC Conveyor.B_RunConveyor_Speed_Max, 100 ms
   "Conveyor_B_Calib_OK" : Bool = PLC Conveyor.B_Calib_OK, 100 ms
   "Conveyor_O_Analog_Value" : Int = PLC Conveyor.O_Analog, 100 ms
   "Temperature_Top_PV_Temper" : Int = PLC Temperature_Top.PV_Temper, 100 ms
   "Temperature_Top_B_Calib_Dim_Point_1" : Bool = PLC Temperature_Top.B_Calib_Dim_Point_1, 100 ms
   "Temperature_Top_B_Calib_Dim_Point_2" : Bool = PLC Temperature_Top.B_Calib_Dim_Point_2, 100 ms
   "Temperature_Top_B_Calib_OK" : Bool = PLC Temperature_Top.B_Calib_OK, 100 ms
   "Temperature_Top_B_Default" : Bool = PLC Temperature_Top.B_Default, 100 ms
   "Temperature_Top_Calib_Enable" : Bool = PLC Temperature_Top.Calib_Enable, 100 ms
   "Temperature_Top_I_Analog_Read" : Int = PLC Temperature_Top.I_Analog_Read, 100 ms
   "Temperature_Top_Calib_Result" : Bool = PLC Temperature_Top.Calib_Result, 100 ms
   "Temperature_Top_SV_Point_1_Temper" : Int = PLC Temperature_Top.SV_Point_1_Temper, 100 ms
   "Temperature_Top_SV_Point_2_Temper" : Int = PLC Temperature_Top.SV_Point_2_Temper, 100 ms
   "Temperature_Top_SV_Temper" : Int = PLC Temperature_Top.SV_Temper, 100 ms
   "Conveyor_O_Result" : Bool = PLC Conveyor.O_Calib_Result, 100 ms
   "Conveyor_B_Default" : Bool = PLC Conveyor.B_Calib_Default, 100 ms
   "PID_Temp_1_ErrorBits" : DWord = PLC PID_Temp_1.ErrorBits, 100 ms
   "Conveyor_H_PID_State" : Int = PLC Conveyor.H_PID_State, 100 ms
   "Conveyor_H_Run_Kp" : Real = PLC Conveyor.H_Run_Kp, 100 ms
   "Conveyor_H_Run_Ki" : Real = PLC Conveyor.H_Run_Ki, 100 ms
   "Conveyor_H_Run_Kd" : Real = PLC Conveyor.H_Run_Kd, 100 ms
   "Conveyor_H_Stop_Kp" : Real = PLC Conveyor.H_Stop_Kp, 100 ms
   "Conveyor_H_Stop_Ki" : Real = PLC Conveyor.H_Stop_Ki, 100 ms
   "Conveyor_H_Stop_Kd" : Real = PLC Conveyor.H_Stop_Kd, 100 ms
   "Conveyor_B_PID_Default" : Bool = PLC Conveyor.B_PID_Default, 100 ms
   "PID_Temp_1_Retain_CtrlParams_Cycle" : Real = PLC PID_Temp_1.Retain.CtrlParams.Cycle, 100 ms
   "PID_Temp_1_State" : Int = PLC PID_Temp_1.State, 100 ms
   "Blister_Show_Total_Row" : Int = PLC Blister_Show.Total_Row, 100 ms
   "Blister_Show_Total_Blister_Column" : Int = PLC Blister_Show.Total_Blister_Column, 100 ms
   "Blister_Show_Arr{0}" : Int = PLC Blister_Show.Arr[0], 100 ms
   "Blister_Animation_Blister_1{0}" : Word = PLC Blister_Animation.Blister_1[0], 100 ms
   "ScreenWidth" : Int AT %DB1.DBW0
   "Blister_Show_Arr" : Array [0..10] of Int = PLC Blister_Show.Arr, 100 ms
   "Blister_Show_Total_Blister_Column_Temp" : Int = PLC Blister_Show.Total_Blister_Column_Temp, 100 ms
   "Forming_Aplice_DB_Sensor" : Bool = PLC Forming_Aplice_DB.Sensor, 100 ms
   "Blister_Animation_Blister_1{1}" : Word = PLC Blister_Animation.Blister_1[1], 100 ms
   "Blister_Animation_Blister_1{2}" : Word = PLC Blister_Animation.Blister_1[2], 100 ms
   "Blister_Animation_Blister_1{3}" : Word = PLC Blister_Animation.Blister_1[3], 100 ms
   "Blister_Animation_Blister_1{4}" : Word = PLC Blister_Animation.Blister_1[4], 100 ms
   "Blister_Animation_Blister_1{5}" : Word = PLC Blister_Animation.Blister_1[5], 100 ms
   "Blister_Animation_Blister_1{6}" : Word = PLC Blister_Animation.Blister_1[6], 100 ms
   "Blister_Animation_Blister_1{7}" : Word = PLC Blister_Animation.Blister_1[7], 100 ms
   "Blister_Animation_Blister_1{8}" : Word = PLC Blister_Animation.Blister_1[8], 100 ms
   "Blister_Animation_Blister_1{9}" : Word = PLC Blister_Animation.Blister_1[9], 100 ms
   "Blister_Animation_Blister_1{10}" : Word = PLC Blister_Animation.Blister_1[10], 100 ms
   "Blister_Animation_Blister_1{11}" : Word = PLC Blister_Animation.Blister_1[11], 100 ms
   "Blister_Animation_Blister_1{12}" : Word = PLC Blister_Animation.Blister_1[12], 100 ms
   "Blister_Animation_Blister_1{13}" : Word = PLC Blister_Animation.Blister_1[13], 100 ms
   "Blister_Animation_Blister_1{14}" : Word = PLC Blister_Animation.Blister_1[14], 100 ms
   "Blister_Animation_Blister_1{15}" : Word = PLC Blister_Animation.Blister_1[15], 100 ms
   "Blister_Animation_Blister_1{16}" : Word = PLC Blister_Animation.Blister_1[16], 100 ms
   "Blister_Animation_Blister_1{17}" : Word = PLC Blister_Animation.Blister_1[17], 100 ms
   "Blister_Animation_Blister_1{18}" : Word = PLC Blister_Animation.Blister_1[18], 100 ms
   "Blister_Animation_Blister_1{19}" : Word = PLC Blister_Animation.Blister_1[19], 100 ms
   "Blister_Animation_Blister_1{20}" : Word = PLC Blister_Animation.Blister_1[20], 100 ms
   "Machine_Data_Angle" : Int = PLC Machine_Data.Angle, 100 ms
   "Enable" : Bool = PLC Enable AT %M0.5, 100 ms
   "Forming_Enable" : Bool = PLC Forming_Enable AT %M0.7, 100 ms
   "Forming_Trig" : Bool = PLC Forming_Trig AT %M0.6, 100 ms
   "Station_Position_Cut_to_ApliceALU" : Int = PLC Station_Position.Cut_to_ApliceALU, 100 ms
   "Station_Position_Cut_to_Camera" : Int = PLC Station_Position.Cut_to_Camera, 100 ms
   "Station_Position_Cut_to_Matrix_Feeder" : Int = PLC Station_Position.Cut_to_Matrix_Feeder, 100 ms
   "Station_Position_Cut_to_PinHole" : Int = PLC Station_Position.Cut_to_PinHole, 100 ms
   "Station_Position_Cut_to_Forming" : Int = PLC Station_Position.Cut_to_Forming, 100 ms
   "Servo_Pull_CW_Trig" : Bool = PLC Servo_Pull_CW_Trig AT %M1.2, 100 ms
   "Servo_Pull_Enable" : Bool = PLC Servo_Pull_Enable AT %M1.0, 100 ms
   "PinHole_Detect" : Bool = PLC PinHole_Detect AT %M1.3, 100 ms
   "Machine_Data_SV_Machine_Speed" : Int = PLC Machine_Data.SV_Machine_Speed, 100 ms
   "Forming_Module_DB_Forming_Switch" : Bool = PLC Forming_Module_DB.Forming_Switch, 100 ms
   "Forming_Module_DB_Forming_Trig" : Bool = PLC Forming_Module_DB.Forming_Trig, 100 ms
   "Forming_Module_DB_SV_Angle_Forming_Begin" : Int = PLC Forming_Module_DB.SV_Angle_Forming_Begin, 100 ms
   "Forming_Module_DB_SV_Angle_Forming_End" : Int = PLC Forming_Module_DB.SV_Angle_Forming_End, 100 ms
   "Matrix_Feeder_DB_Switch_on/off" : Bool = PLC Matrix_Feeder_DB.Switch_on/off, 100 ms
   "Matrix_Feeder_DB_I_Step_Feeder" : Int = PLC Matrix_Feeder_DB.I_Step_Feeder, 100 ms
   "Matrix_Feeder_DB_Q_Feeder" : Bool = PLC Matrix_Feeder_DB.Q_Feeder, 100 ms
   "Matrix_Feeder_DB_Angel_Begin" : Int = PLC Matrix_Feeder_DB.Angel_Begin, 100 ms
   "Matrix_Feeder_DB_Angel_End" : Int = PLC Matrix_Feeder_DB.Angel_End, 100 ms
   "Step" : Int = PLC Step AT %MW52, 1 s
   "Blister_Animation_Blister_Matrix{0}" : Word = PLC Blister_Animation.Blister_Matrix[0], 100 ms
   "Blister_Animation_Blister_Matrix{1}" : Word = PLC Blister_Animation.Blister_Matrix[1], 100 ms
   "Blister_Animation_Blister_Matrix{2}" : Word = PLC Blister_Animation.Blister_Matrix[2], 100 ms
   "Blister_Animation_Blister_Matrix{20}" : Word = PLC Blister_Animation.Blister_Matrix[20], 100 ms
   "Blister_Animation_Blister_Matrix{19}" : Word = PLC Blister_Animation.Blister_Matrix[19], 100 ms
   "Blister_Animation_Blister_Matrix{18}" : Word = PLC Blister_Animation.Blister_Matrix[18], 100 ms
   "Blister_Animation_Blister_Matrix{17}" : Word = PLC Blister_Animation.Blister_Matrix[17], 100 ms
   "Blister_Animation_Blister_Matrix{16}" : Word = PLC Blister_Animation.Blister_Matrix[16], 100 ms
   "Blister_Animation_Blister_Matrix{15}" : Word = PLC Blister_Animation.Blister_Matrix[15], 100 ms
   "Blister_Animation_Blister_Matrix{14}" : Word = PLC Blister_Animation.Blister_Matrix[14], 100 ms
   "Blister_Animation_Blister_Matrix{13}" : Word = PLC Blister_Animation.Blister_Matrix[13], 100 ms
   "Blister_Animation_Blister_Matrix{12}" : Word = PLC Blister_Animation.Blister_Matrix[12], 100 ms
   "Blister_Animation_Blister_Matrix{11}" : Word = PLC Blister_Animation.Blister_Matrix[11], 100 ms
   "Blister_Animation_Blister_Matrix{10}" : Word = PLC Blister_Animation.Blister_Matrix[10], 100 ms
   "Blister_Animation_Blister_Matrix{9}" : Word = PLC Blister_Animation.Blister_Matrix[9], 100 ms
   "Blister_Animation_Blister_Matrix{8}" : Word = PLC Blister_Animation.Blister_Matrix[8], 100 ms
   "Blister_Animation_Blister_Matrix{7}" : Word = PLC Blister_Animation.Blister_Matrix[7], 100 ms
   "Blister_Animation_Blister_Matrix{6}" : Word = PLC Blister_Animation.Blister_Matrix[6], 100 ms
   "Blister_Animation_Blister_Matrix{5}" : Word = PLC Blister_Animation.Blister_Matrix[5], 100 ms
   "Blister_Animation_Blister_Matrix{4}" : Word = PLC Blister_Animation.Blister_Matrix[4], 100 ms
   "Blister_Animation_Blister_Matrix{3}" : Word = PLC Blister_Animation.Blister_Matrix[3], 100 ms
   "Batch_Management_DB_Lot_Size" : DInt = PLC Batch_Management_DB.Lot_Size, 1 s
   "Batch_Management_DB_PV_Lot_Status" : USInt = PLC Batch_Management_DB.PV_Lot_Status, 100 ms
   "Batch_Management_DB_B_Start_Lot" : Bool = PLC Batch_Management_DB.B_Start_Lot, 1 s
   "Batch_Management_DB_B_Finish_Lot" : Bool = PLC Batch_Management_DB.B_Finish_Lot, 1 s
   "Batch_Management_DB_PV_Lot_Running_Total_Time" : DInt = PLC Batch_Management_DB.PV_Lot_Running_Total_Time, 1 s
   "Batch_Management_DB_B_Hold_Lot" : Bool = PLC Batch_Management_DB.B_Hold_Lot, 1 s
   "Batch_Management_DB_SV_Sampling_Time" : DInt = PLC Batch_Management_DB.SV_Sampling_Time, 1 s
   "Hide" : Bool AT %DB1.DBW0
   "Batch_Management_DB_Reset_Sampling_Time" : Bool = PLC Batch_Management_DB.Reset_Sampling_Time, 1 s
   "Batch_Management_DB_T_ET" : Time = PLC Batch_Management_DB.T.ET, 1 s
   "Batch_Management_DB_Q_Write_Report" : Bool = PLC Batch_Management_DB.Q_Write_Report, 100 ms
      on ChangeValue: "Write_Report"()
   "Recipe_Data_Data_1" : Int = PLC Recipe_Data.Data_1, 1 s
   "Recipe_Data_Data_2" : Int = PLC Recipe_Data.Data_2, 1 s
   "Recipe_Data_Data_3" : Int = PLC Recipe_Data.Data_3, 1 s
   "Recipe_Data_Data_4" : Int = PLC Recipe_Data.Data_4, 1 s
   "Recipe_Data_Data_5" : Int = PLC Recipe_Data.Data_5, 1 s
   "Batch_Management_DB_Product_Name" : Int = PLC Batch_Management_DB.Product_Name, 1 s
   "Batch_Management_DB_Batch_Number" : Int = PLC Batch_Management_DB.Batch_Number, 1 s
   "Batch_Management_DB_Recipe_Name" : String[254] = PLC Batch_Management_DB.Recipe_Name_1, 1 s
   "Batch_Management_DB_Recipe_Record" : Int = PLC Batch_Management_DB.Recipe_Record_1, 1 s
   "Batch_Management_DB_Trig" : Bool = PLC Batch_Management_DB.Trig, 1 s
   "Batch_Management_DB_Recipe_Name_2" : String[254] = PLC Batch_Management_DB.Recipe_Name_2, 1 s
   "Batch_Management_DB_Recipe_Record_2" : Int = PLC Batch_Management_DB.Recipe_Record_2, 1 s
   "Batch_Management_DB_Trig2" : Bool = PLC Batch_Management_DB.Trig2, 1 s
   "Downloaded" : Bool AT %DB1.DBX0.0
   "Status_Batch" : USInt = PLC Batch_Management_DB.PV_Lot_Status, 1 s
   "Status_Batch_Number" : Int = PLC Batch_Management_DB.Batch_Number AT %DB1.DBB0, 1 s
   "Batch_Management_DB_Record_Number" : Int = PLC Batch_Management_DB.Recipe_Record_1, 1 s
   "Record_Number_Ac" : Int = PLC Batch_Management_DB.Record_Number AT %DB1.DBW0, 1 s

text list "Mode PID": 0 'Tắt'; 1 ''; 2 ''; 3 'Tự động'; 4 'Thủ công'; 5 ''

text list "Lot_Status": 1 'Hold'; 2 'Running'; 0 'Stop'

recipe "Recipe_11": Item_1 <- "Batch_Management_DB_Product_Name", Item_2 <- "Batch_Management_DB_Batch_Number", Item_3 <- "Batch_Management_DB_PV_Lot_Status", Item_4 <- "Batch_Management_DB_Recipe_Record", Item_5 <- "Recipe_Data_Data_5"

screen "Conveyor_Calib" 1024x768, template "Template_1"
   on GenerateScreen: SetBit("Conveyor_Calib_Enable")
   on ClearScreen: ResetBit("Conveyor_Calib_Enable")
   IOField "I/O field_2" at 134,310 size 221x73; FormatPattern 999
      ProcessValue <- "Conveyor_Calib_Speed_1"
   TextField "Text field_1" at 82,221 size 290x90; Text 'Tốc độ băng tải Min'
   IOField "I/O field_1" at 663,310 size 221x73; FormatPattern 999
      ProcessValue <- "Conveyor_Calib_Speed_2"
   TextField "Text field_2" at 629,221 size 290x90; Text 'Tốc độ băng tải Max'
   TextField "Text field_3" at 170,1 size 690x72; Text 'Hiệu chỉnh tốc độ băng tải'
   Switch "Switch_1" at 13,416 size 463x103; CaptionText 'Switch'; TextOff 'Băng tải chạy tốc độ tối thiểu TẮT'; TextOn 'Băng tải chạy tốc độ tối thiểu MỞ'
      ProcessValue <- "Conveyor_B_RunConveyor_Speed_Min"
      Appearance <- "Conveyor_B_RunConveyor_Speed_Min"
   Switch "Switch_2" at 542,416 size 463x103; TextOn 'Băng tải chạy tốc độ tối đa MỞ'; CaptionText 'Switch'; TextOff 'Băng tải chạy tốc độ tối đa TẮT'
      ProcessValue <- "Conveyor_B_RunConveyor_Speed_Max"
      Appearance <- "Conveyor_B_RunConveyor_Speed_Max"
   IOField "I/O field_3" at 351,123 size 221x73; FormatPattern 99999
      ProcessValue <- "Conveyor_O_Analog_Value"
   TextField "Text field_4" at 35,118 size 290x90; Text 'Giá trị Analog out'
   Button "Button_3" at 530,682 size 221x73; TextOff 'OK'
      on Press: SetBit("Conveyor_B_Calib_OK")
      Appearance <- "Conveyor_O_Result"
   TextField "Text field_8" at 394,598 size 237x79; Text 'Thành công'
      Visibility <- "Conveyor_O_Result"
   Button "Button_4" at 271,682 size 221x73; TextOff 'Mặc định'
      on Press: SetBit("Conveyor_B_Default")
   Switch "Switch_3" at 134,530 size 221x73; TextOn 'ON'; CaptionText 'Switch'; TextOff 'OFF'
      ProcessValue <- "Conveyor_Calib_Dim_Point_1"
      Appearance <- "Conveyor_Calib_Dim_Point_1"
   Switch "Switch_4" at 663,530 size 221x73; TextOn 'ON'; CaptionText 'Switch'; TextOff 'OFF'
      ProcessValue <- "Conveyor_Calib_Dim_Point_2"
      Appearance <- "Conveyor_Calib_Dim_Point_2"
   Slider "Slider_1" at 916,74 size 70x241; Caption 'SIMATIC'
      ProcessValue <- "Conveyor_O_Analog_Value"

screen "Calib_Temper_Top" 1024x768, template "Template_1"
   on GenerateScreen: SetBit("Temperature_Top_Calib_Enable")
   on ClearScreen: ResetBit("Temperature_Top_Calib_Enable")
   TextField "Text field_3" at 170,1 size 690x67; Text 'Hiệu chỉnh nhiệt độ trên'
   IOField "I/O field_3" at 351,88 size 221x73; FormatPattern 99999
      ProcessValue <- "Temperature_Top_I_Analog_Read"
   TextField "Text field_4" at 35,83 size 290x90; Text 'Giá trị Analog in'
   Button "Button_3" at 529,682 size 221x73; TextOff 'OK'
      on Press: SetBit("Temperature_Top_B_Calib_OK")
      Appearance <- "Temperature_Top_Calib_Result"
   TextField "Text field_5" at 34,163 size 290x90; Text 'Nhiệt độ đặt'
   IOField "I/O field_4" at 350,171 size 221x73; FormatPattern 999
      ProcessValue <- "Temperature_Top_SV_Temper"
   TextField "Text field_6" at 587,168 size 111x79; Text '(độ C)'
   Button "Button_4" at 271,682 size 221x73; TextOff 'Mặc định'
      on Press: SetBit("Temperature_Top_B_Default")
   TextField "Text field_1" at 118,351 size 290x77; Text 'Nhiệt độ môi trường'
   IOField "I/O field_2" at 152,447 size 221x73; FormatPattern 999
      ProcessValue <- "Temperature_Top_SV_Point_1_Temper"
   TextField "Text field_2" at 576,345 size 290x90; Text 'Nhiệt độ làm việc'
   IOField "I/O field_1" at 610,447 size 221x73; FormatPattern 999
      ProcessValue <- "Temperature_Top_SV_Point_2_Temper"
   TextField "Text field_8" at 394,598 size 237x79; Text 'Thành công'
      Visibility <- "Temperature_Top_Calib_Result"
   TextField "Text field_7" at 34,247 size 290x90; Text 'Nhiệt độ hiện tại'
   IOField "I/O field_5" at 350,255 size 221x73; FormatPattern 999
      ProcessValue <- "Temperature_Top_PV_Temper"
   TextField "Text field_9" at 587,247 size 111x79; Text '(độ C)'
   TextField "Text field_10" at 380,441 size 111x79; Text '(độ C)'
   TextField "Text field_11" at 846,441 size 111x79; Text '(độ C)'
   Slider "Slider_1" at 808,85 size 70x241; Caption 'SIMATIC'
      ProcessValue <- "Temperature_Top_I_Analog_Read"
   Slider "Slider_2" at 926,85 size 70x241; Caption 'SIMATIC'
      ProcessValue <- "Temperature_Top_PV_Temper"
   Switch "Switch_1" at 152,534 size 221x73; CaptionText 'Switch'; TextOff 'OFF'; TextOn 'ON'
      ProcessValue <- "Temperature_Top_B_Calib_Dim_Point_1"
      Appearance <- "Temperature_Top_B_Calib_Dim_Point_1"
   Switch "Switch_2" at 610,534 size 221x73; TextOn 'ON'; CaptionText 'Switch'; TextOff 'OFF'
      ProcessValue <- "Temperature_Top_B_Calib_Dim_Point_2"
      Appearance <- "Temperature_Top_B_Calib_Dim_Point_2"

screen "Calib" 1024x768
   TextField "Text field_3" at 170,22 size 690x90; Text 'Hiệu chỉnh'
   Button "Button_3" at 115,112 size 284x73; TextOff 'Tốc độ băng tải'
      on Press: ActivateScreen("Conveyor_Calib", 0)
   Button "Button_1" at 115,213 size 284x73; TextOff 'Nhiệt trên'
      on Press: ActivateScreen("Calib_Temper_Top", 0)
   Button "Button_2" at 115,309 size 284x73; TextOff 'PID Nhiệt trên'
      on Press: ActivateScreen("PID_Setting", 0)

Template "Template_1" 1024x768
   Button "Button_3" at 12,682 size 221x73; TextOff 'Trở về'
      on Press: function_efd93a16()

screen "PID_Setting" 1024x768, template "Template_1"
   IOField "I/O field_2" at 127,353 size 174x60; FormatPattern 99.9
      ProcessValue <- "Conveyor_H_Stop_Kp"
   TextField "Text field_1" at 279,4 size 432x67; Text 'Cài đặt PID nhiệt trên'
   TextField "Text field_2" at 27,146 size 150x67; Text 'Chế độ'
   SymbolicIOField "Symbolic I/O field_1" at 197,156 size 223x47; TextOff '0'; TextOn '1'; TextList "Mode PID"
      ProcessValue <- "Conveyor_H_PID_State"
   IOField "I/O field_4" at 759,95 size 129x47; FormatPattern FFFF
      ProcessValue <- "PID_Temp_1_ErrorBits"
   TextField "Text field_3" at 577,85 size 150x67; Text 'Mã lỗi'
   TextField "Text field_4" at 27,350 size 150x67; Text 'Kp'
   TextField "Text field_5" at 79,282 size 271x67; Text 'Khi máy dừng'
   TextField "Text field_6" at 28,412 size 150x67; Text 'Ki'
   TextField "Text field_7" at 27,475 size 150x67; Text 'Kd'
   IOField "I/O field_6" at 127,415 size 174x60; FormatPattern 99.9
      ProcessValue <- "Conveyor_H_Stop_Ki"
   IOField "I/O field_7" at 127,478 size 174x60; FormatPattern 99.9
      ProcessValue <- "Conveyor_H_Stop_Kd"
   IOField "I/O field_1" at 364,353 size 174x60; FormatPattern 99.9
      ProcessValue <- "Conveyor_H_Run_Kp"
   TextField "Text field_8" at 316,282 size 271x67; Text 'Khi máy chạy'
   IOField "I/O field_9" at 364,415 size 174x60; FormatPattern 99.9
      ProcessValue <- "Conveyor_H_Run_Ki"
   IOField "I/O field_10" at 364,478 size 174x60; FormatPattern 99.9
      ProcessValue <- "Conveyor_H_Run_Kd"
   IOField "I/O field_5" at 820,503 size 174x60; FormatPattern 999
      ProcessValue <- "PID_Temp_1_Retain_CtrlParams_Cycle"
   TextField "Text field_9" at 577,500 size 271x67; Text 'Chu kỳ lấy mẫu'
   TextField "Text field_10" at 27,213 size 150x67; Text 'Chế độ'
   SymbolicIOField "Symbolic I/O field_2" at 197,223 size 223x47; TextOn '1'; TextOff '0'; TextList "Mode PID"
   Button "Button_4" at 271,682 size 221x73; TextOff 'Mặc định'
      on Press: SetBit("Conveyor_B_PID_Default")
   TextField "Text field_11" at 27,85 size 156x67; Text 'Trạng thái:'
   Button "Button_1" at 199,95 size 198x47; TextOff 'Text'; TextList "Mode PID"
      ProcessValue <- "PID_Temp_1_State"

screen "Blister_Setting" 1024x768
   on GenerateScreen: "Total_Blister_test"()
   Rectangle "BlisterRow_6" at 964,546 size 41x11
      Appearance <- "Blister_Animation_Blister_1{0}"
      Visibility <- "Blister_Show_Total_Row"
   Rectangle "BlisterRow_5" at 964,560 size 41x11
      Appearance <- "Blister_Animation_Blister_1{0}"
      Visibility <- "Blister_Show_Total_Row"
   Rectangle "BlisterRow_4" at 964,575 size 41x11
      Appearance <- "Blister_Animation_Blister_1{0}"
      Visibility <- "Blister_Show_Total_Row"
   Rectangle "BlisterRow_3" at 964,590 size 41x11
      Appearance <- "Blister_Animation_Blister_1{0}"
      Visibility <- "Blister_Show_Total_Row"
   Rectangle "BlisterRow_2" at 964,605 size 41x11
      Appearance <- "Blister_Animation_Blister_1{0}"
      Visibility <- "Blister_Show_Total_Row"
   Rectangle "BlisterRow_1" at 964,620 size 41x11
      Appearance <- "Blister_Animation_Blister_1{0}"
      Visibility <- "Blister_Show_Total_Row"
   Rectangle "Blister_7" at 54,546 size 23x85
      Visibility <- "Blister_Show_Total_Blister_Column"
      Appearance <- "Blister_Animation_Blister_1{7}"
   Rectangle "Blister_1" at 54,546 size 23x85
      Visibility <- "Blister_Show_Total_Blister_Column"
      Appearance <- "Blister_Animation_Blister_1{1}"
   Rectangle "Blister_2" at 54,546 size 23x85
      Visibility <- "Blister_Show_Total_Blister_Column"
      Appearance <- "Blister_Animation_Blister_1{2}"
   Rectangle "Blister_3" at 54,546 size 23x85
      Visibility <- "Blister_Show_Total_Blister_Column"
      Appearance <- "Blister_Animation_Blister_1{3}"
   Rectangle "Blister_4" at 54,546 size 23x85
      Visibility <- "Blister_Show_Total_Blister_Column"
      Appearance <- "Blister_Animation_Blister_1{4}"
   Rectangle "Blister_5" at 54,546 size 23x85
      Visibility <- "Blister_Show_Total_Blister_Column"
      Appearance <- "Blister_Animation_Blister_1{5}"
   Rectangle "Blister_6" at 54,546 size 23x85
      Visibility <- "Blister_Show_Total_Blister_Column"
      Appearance <- "Blister_Animation_Blister_1{6}"
   Rectangle "Blister_8" at 54,546 size 23x85
      Visibility <- "Blister_Show_Total_Blister_Column"
      Appearance <- "Blister_Animation_Blister_1{8}"
   Rectangle "Blister_9" at 54,546 size 23x85
      Visibility <- "Blister_Show_Total_Blister_Column"
      Appearance <- "Blister_Animation_Blister_1{9}"
   Rectangle "Blister_10" at 54,546 size 23x85
      Visibility <- "Blister_Show_Total_Blister_Column"
      Appearance <- "Blister_Animation_Blister_1{10}"
   IOField "I/O field_5" at 111,724 size 96x32; FormatPattern 99
      ProcessValue <- "Blister_Show_Total_Blister_Column_Temp"
   TextField "Text field_1" at 10,729 size 60x22; Text 'Column'
   Rectangle "Blister_11" at 54,546 size 23x85
      Visibility <- "Blister_Show_Total_Blister_Column"
      Appearance <- "Blister_Animation_Blister_1{11}"
   Rectangle "Blister_12" at 54,546 size 23x85
      Visibility <- "Blister_Show_Total_Blister_Column"
      Appearance <- "Blister_Animation_Blister_1{12}"
   Rectangle "Blister_13" at 54,546 size 23x85
      Visibility <- "Blister_Show_Total_Blister_Column"
      Appearance <- "Blister_Animation_Blister_1{13}"
   Rectangle "Blister_14" at 54,546 size 23x85
      Visibility <- "Blister_Show_Total_Blister_Column"
      Appearance <- "Blister_Animation_Blister_1{14}"
   Rectangle "Blister_15" at 54,546 size 23x85
      Visibility <- "Blister_Show_Total_Blister_Column"
      Appearance <- "Blister_Animation_Blister_1{15}"
   Rectangle "Blister_16" at 54,546 size 23x85
      Visibility <- "Blister_Show_Total_Blister_Column"
      Appearance <- "Blister_Animation_Blister_1{16}"
   Rectangle "Blister_17" at 54,546 size 23x85
      Visibility <- "Blister_Show_Total_Blister_Column"
      Appearance <- "Blister_Animation_Blister_1{17}"
   Rectangle "Blister_18" at 54,546 size 23x85
      Visibility <- "Blister_Show_Total_Blister_Column"
      Appearance <- "Blister_Animation_Blister_1{18}"
   Rectangle "Blister_19" at 54,546 size 23x85
      Visibility <- "Blister_Show_Total_Blister_Column"
      Appearance <- "Blister_Animation_Blister_1{19}"
   Rectangle "Blister_20" at 54,546 size 23x85
      Visibility <- "Blister_Show_Total_Blister_Column"
      Appearance <- "Blister_Animation_Blister_1{20}"
   Button "Button_2" at 439,510 size 143x32; TextOff 'PinHole Detetct'
      on Press: SetBit("PinHole_Detect")
      on Release: ResetBit("PinHole_Detect")
   Button "Button_4" at 886,444 size 96x32; TextOff 'Matrix'
      on Press: "Total_Blister"()
   Button "Button_5" at 456,228 size 96x32; TextOff 'Camera'
      on Press: "Total_Blister"()
   Button "Button_6" at 456,722 size 51x32; TextOff 'Nối'
   IOField "I/O field_2" at 111,672 size 96x32; FormatPattern 9
      ProcessValue <- "Blister_Show_Total_Row"
   TextField "Text field_2" at 10,677 size 82x22; Text 'Số hàng vỉ'
   IOField "I/O field_4" at 864,198 size 141x32; FormatPattern 111111
      ProcessValue <- "Blister_Animation_Blister_1{1}"
   Gauge "Gauge_1" at 879,9 size 103x103; CaptionText 'SIMATIC'; UnitText 'Unit'
      ProcessValue <- "Machine_Data_Angle"
   IOField "I/O field_6" at 593,617 size 87x32; FormatPattern 111111
      ProcessValue <- "Blister_Animation_Blister_Matrix{17}"
   IOField "I/O field_7" at 593,582 size 87x32; FormatPattern 111111
      ProcessValue <- "Blister_Animation_Blister_Matrix{16}"
   IOField "I/O field_8" at 593,547 size 87x32; FormatPattern 111111
      ProcessValue <- "Blister_Animation_Blister_Matrix{15}"
   IOField "I/O field_9" at 593,511 size 87x32; FormatPattern 111111
      ProcessValue <- "Blister_Animation_Blister_Matrix{14}"
   IOField "I/O field_10" at 593,476 size 87x32; FormatPattern 111111
      ProcessValue <- "Blister_Animation_Blister_Matrix{13}"
   IOField "I/O field_11" at 593,441 size 87x32; FormatPattern 111111
      ProcessValue <- "Blister_Animation_Blister_Matrix{12}"
   IOField "I/O field_15" at 593,299 size 87x32; FormatPattern 111111
      ProcessValue <- "Blister_Animation_Blister_Matrix{8}"
   IOField "I/O field_16" at 593,264 size 87x32; FormatPattern 111111
      ProcessValue <- "Blister_Animation_Blister_Matrix{7}"
   IOField "I/O field_17" at 593,229 size 87x32; FormatPattern 111111
      ProcessValue <- "Blister_Animation_Blister_Matrix{6}"
   IOField "I/O field_18" at 593,193 size 87x32; FormatPattern 111111
      ProcessValue <- "Blister_Animation_Blister_Matrix{5}"
   IOField "I/O field_19" at 593,158 size 87x32; FormatPattern 111111
      ProcessValue <- "Blister_Animation_Blister_Matrix{4}"
   IOField "I/O field_20" at 593,123 size 87x32; FormatPattern 111111
      ProcessValue <- "Blister_Animation_Blister_Matrix{3}"
   IOField "I/O field_21" at 593,87 size 87x32; FormatPattern 111111
      ProcessValue <- "Blister_Animation_Blister_Matrix{2}"
   IOField "I/O field_22" at 593,52 size 87x32; FormatPattern 111111
      ProcessValue <- "Blister_Animation_Blister_Matrix{1}"
   IOField "I/O field_24" at 593,653 size 87x32; FormatPattern 111111
      ProcessValue <- "Blister_Animation_Blister_Matrix{18}"
   IOField "I/O field_25" at 593,688 size 87x32; FormatPattern 111111
      ProcessValue <- "Blister_Animation_Blister_Matrix{19}"
   IOField "I/O field_26" at 593,724 size 87x32; FormatPattern 111111
      ProcessValue <- "Blister_Animation_Blister_Matrix{20}"
   TextField "Text field_3" at 703,730 size 25x22; Text '20'
   TextField "Text field_4" at 703,376 size 25x22; Text '10'
   TextField "Text field_5" at 703,56 size 15x22; Text '1'
   IOField "I/O field_23" at 593,9 size 87x32; FormatPattern 111111
      ProcessValue <- "Blister_Animation_Blister_1{0}"
   Switch "Switch_2" at 456,599 size 86x51; TextOn 'ON'; CaptionText 'Forming'; TextOff 'OFF'
      ProcessValue <- "Forming_Module_DB_Forming_Switch"
   Circle "Circle_1" at 552,618 size 30x30
      Appearance <- "Forming_Module_DB_Forming_Trig"
   TextField "Text field_6" at 11,12 size 258x29; Text 'KC Forming đến dao cắt'
   TextField "Text field_7" at 11,47 size 258x29; Text 'KC PinHole đến dao cắt'
   TextField "Text field_8" at 11,83 size 258x29; Text 'KC Matrix đến dao cắt'
   TextField "Text field_9" at 11,118 size 258x29; Text 'KC Camera đến dao cắt'
   TextField "Text field_10" at 11,154 size 258x29; Text 'KC nối ALU đến dao cắt'
   IOField "I/O field_1" at 268,152 size 56x32; FormatPattern 99
      ProcessValue <- "Station_Position_Cut_to_ApliceALU"
   IOField "I/O field_27" at 268,116 size 56x32; FormatPattern 99
      ProcessValue <- "Station_Position_Cut_to_Camera"
   IOField "I/O field_28" at 268,81 size 56x32; FormatPattern 99
      ProcessValue <- "Station_Position_Cut_to_Matrix_Feeder"
   IOField "I/O field_29" at 268,45 size 56x32; FormatPattern 99
      ProcessValue <- "Station_Position_Cut_to_PinHole"
   IOField "I/O field_30" at 268,10 size 56x32; FormatPattern 99
      ProcessValue <- "Station_Position_Cut_to_Forming"
   Circle "Circle_2" at 910,311 size 30x30
      Appearance <- "Servo_Pull_CW_Trig"
   TextField "Text field_11" at 860,315 size 33x22; Text 'Kéo'
   Switch "Switch_3" at 864,250 size 86x51; TextOn 'ON'; CaptionText 'Kéo'; TextOff 'OFF'
      ProcessValue <- "Servo_Pull_Enable"
   Button "Button_3" at 250,672 size 109x32; TextOff 'Animation'
      on Press: "Total_Blister_test"()
   TextField "Text field_12" at 703,554 size 25x22; Text '15'
   TextField "Text field_13" at 700,198 size 15x22; Text '5'
   TextField "Text field_14" at 11,201 size 258x29; Text 'Góc Forming'
   IOField "I/O field_32" at 268,196 size 56x32; FormatPattern 999
      ProcessValue <- "Forming_Module_DB_SV_Angle_Forming_Begin"
   IOField "I/O field_33" at 341,196 size 56x32; FormatPattern 999
      ProcessValue <- "Forming_Module_DB_SV_Angle_Forming_End"
   TextField "Text field_15" at 11,245 size 258x29; Text 'Góc Matrix'
   TextField "Text field_16" at 11,289 size 258x29; Text 'Góc Camera'
   Rectangle "Rectangle_1" at 570,367 size 133x37
      Appearance <- "Matrix_Feeder_DB_Q_Feeder"
   IOField "I/O field_34" at 496,10 size 56x32; FormatPattern 99
      ProcessValue <- "Matrix_Feeder_DB_I_Step_Feeder"
   TextField "Text field_17" at 330,12 size 137x29; Text 'Bước cấp viên'
   Switch "Switch_1" at 460,352 size 86x51; TextOn 'ON'; CaptionText 'Matrix Feeder'; TextOff 'OFF'
      ProcessValue <- "Matrix_Feeder_DB_Switch_on/off"
   IOField "I/O field_35" at 268,242 size 56x32; FormatPattern 999
      ProcessValue <- "Matrix_Feeder_DB_Angel_Begin"
   IOField "I/O field_36" at 341,242 size 56x32; FormatPattern 999
      ProcessValue <- "Matrix_Feeder_DB_Angel_End"
   Rectangle "Rectangle_2" at 570,403 size 133x37
      Appearance <- "Matrix_Feeder_DB_Q_Feeder"
      Visibility <- "Matrix_Feeder_DB_I_Step_Feeder"
   IOField "I/O field_37" at 460,315 size 96x32; FormatPattern 9
      ProcessValue <- "Step"
   IOField "I/O field_38" at 731,616 size 87x32; FormatPattern 111111
      ProcessValue <- "Blister_Animation_Blister_1{17}"
   IOField "I/O field_39" at 731,581 size 87x32; FormatPattern 111111
      ProcessValue <- "Blister_Animation_Blister_1{16}"
   IOField "I/O field_40" at 731,546 size 87x32; FormatPattern 111111
      ProcessValue <- "Blister_Animation_Blister_1{15}"
   IOField "I/O field_41" at 731,510 size 87x32; FormatPattern 111111
      ProcessValue <- "Blister_Animation_Blister_1{14}"
   IOField "I/O field_42" at 731,475 size 87x32; FormatPattern 111111
      ProcessValue <- "Blister_Animation_Blister_1{13}"
   IOField "I/O field_43" at 731,440 size 87x32; FormatPattern 111111
      ProcessValue <- "Blister_Animation_Blister_1{12}"
   IOField "I/O field_44" at 731,298 size 87x32; FormatPattern 111111
      ProcessValue <- "Blister_Animation_Blister_1{8}"
   IOField "I/O field_45" at 731,263 size 87x32; FormatPattern 111111
      ProcessValue <- "Blister_Animation_Blister_1{7}"
   IOField "I/O field_46" at 731,228 size 87x32; FormatPattern 111111
      ProcessValue <- "Blister_Animation_Blister_1{6}"
   IOField "I/O field_47" at 731,192 size 87x32; FormatPattern 111111
      ProcessValue <- "Blister_Animation_Blister_1{5}"
   IOField "I/O field_48" at 731,157 size 87x32; FormatPattern 111111
      ProcessValue <- "Blister_Animation_Blister_1{4}"
   IOField "I/O field_49" at 731,122 size 87x32; FormatPattern 111111
      ProcessValue <- "Blister_Animation_Blister_1{3}"
   IOField "I/O field_50" at 731,86 size 87x32; FormatPattern 111111
      ProcessValue <- "Blister_Animation_Blister_1{2}"
   IOField "I/O field_51" at 731,51 size 87x32; FormatPattern 111111
      ProcessValue <- "Blister_Animation_Blister_1{1}"
   IOField "I/O field_52" at 731,652 size 87x32; FormatPattern 111111
      ProcessValue <- "Blister_Animation_Blister_1{18}"
   IOField "I/O field_53" at 731,687 size 87x32; FormatPattern 111111
      ProcessValue <- "Blister_Animation_Blister_1{19}"
   IOField "I/O field_54" at 731,723 size 87x32; FormatPattern 111111
      ProcessValue <- "Blister_Animation_Blister_1{20}"
   IOField "I/O field_58" at 731,9 size 87x32; FormatPattern 111111
      ProcessValue <- "Blister_Animation_Blister_1{0}"
   IOField "I/O field_3" at 903,67 size 51x24; FormatPattern 999
      ProcessValue <- "Machine_Data_Angle"
   IOField "I/O field_31" at 964,67 size 51x24; FormatPattern 999
      ProcessValue <- "Machine_Data_SV_Machine_Speed"
   IOField "I/O field_14" at 593,335 size 87x32; FormatPattern 111111
      ProcessValue <- "Blister_Animation_Blister_Matrix{9}"
   IOField "I/O field_13" at 593,370 size 87x32; FormatPattern 111111
      ProcessValue <- "Blister_Animation_Blister_Matrix{10}"
   IOField "I/O field_12" at 593,405 size 87x32; FormatPattern 111111
      ProcessValue <- "Blister_Animation_Blister_Matrix{11}"
   IOField "I/O field_55" at 731,334 size 87x32; FormatPattern 111111
      ProcessValue <- "Blister_Animation_Blister_1{9}"
   IOField "I/O field_56" at 731,369 size 87x32; FormatPattern 111111
      ProcessValue <- "Blister_Animation_Blister_1{10}"
   IOField "I/O field_57" at 731,404 size 87x32; FormatPattern 111111
      ProcessValue <- "Blister_Animation_Blister_1{11}"

screen "Batch_Management" 1024x768
   IOField "I/O field_32" at 284,296 size 432x38; FormatPattern s99999
      ProcessValue <- "Batch_Management_DB_Product_Name"
      ObjectEnable <- "Status_Batch"
   TextField "Text field_14" at 14,296 size 177x29; Text 'Tên sản phẩm'
   TextField "Text field_1" at 14,347 size 177x29; Text 'Số lô'
   TextField "Text field_2" at 14,389 size 177x29; Text 'Cở lô'
   Button "start" at 41,652 size 124x85; TextOff 'Bắt đầu lô'
      on Press: "Check_Lot"(); function_bbf3fe93(1, N)
      Visibility <- "Batch_Management_DB_PV_Lot_Status"
   Button "end" at 485,654 size 124x85; TextOff 'Kết thúc lô'
      on Press: SetBit("Batch_Management_DB_B_Finish_Lot"); function_b456aad1("Recipe_11", N); function_f38ba6b2(1, "Record_Number_Ac", 1, 0, N)
      Visibility <- "Batch_Management_DB_PV_Lot_Status"
   Button "Button_2" at 767,654 size 124x85; TextOff 'Tìm kiếm lô'
      on Press: "Total_Blister"()
   IOField "I/O field_1" at 284,337 size 432x38; FormatPattern s99999
      ProcessValue <- "Batch_Management_DB_Batch_Number"
      ObjectEnable <- "Status_Batch"
   IOField "I/O field_2" at 284,377 size 432x38; FormatPattern 9999999999
      ProcessValue <- "Batch_Management_DB_Lot_Size"
      ObjectEnable <- "Batch_Management_DB_PV_Lot_Status"
   TextField "Text field_4" at 14,430 size 177x29; Text 'Bắt đầu'
   IOField "I/O field_3" at 284,418 size 432x38; FormatPattern 9999999999999999999999999999999999999999
   TextField "Text field_5" at 14,473 size 177x29; Text 'Kết thúc'
   TextField "Text field_6" at 14,506 size 177x29; Text 'Thời gian chạy'
   IOField "I/O field_5" at 284,502 size 432x38; FormatPattern 99999
      ProcessValue <- "Batch_Management_DB_PV_Lot_Running_Total_Time"
   IOField "I/O field_6" at 284,546 size 432x38; FormatPattern 9999999999
      ProcessValue <- "Batch_Management_DB_SV_Sampling_Time"
      on OnFinishInput: SetBit("Batch_Management_DB_Reset_Sampling_Time")
   IOField "I/O field_4" at 284,461 size 432x38; FormatPattern 9999999999999999999999999999999999999999
   TextField "Text field_7" at 13,546 size 292x39; Text 'Thời gian lấy mẫu report'
   RecipeView "Recipe view_1" at 2,83 size 791x136; Tag4DataRecord "Batch_Management_DB_Recipe_Record"; Recipe "Recipe_11"
   Button "Pause" at 191,654 size 124x85; TextOff 'Tạm dừng'
      on Press: SetTag("Batch_Management_DB_PV_Lot_Status", 1); function_b456aad1("Recipe_11", N); function_f38ba6b2(1, "Batch_Management_DB_Recipe_Record", 1, 1, N)
      Visibility <- "Batch_Management_DB_PV_Lot_Status"
   Button "Continuous" at 335,654 size 124x85; TextOff 'Tiếp tục'
      on Press: function_bbf3fe93(1, N); SetTag("Batch_Management_DB_PV_Lot_Status", 2)
      Visibility <- "Batch_Management_DB_PV_Lot_Status"
   IOField "I/O field_7" at 16,600 size 96x32; FormatPattern s99999
      ProcessValue <- "Batch_Management_DB_Product_Name"
   IOField "I/O field_8" at 165,603 size 96x32; FormatPattern s99999
      ProcessValue <- "Batch_Management_DB_Batch_Number"
   IOField "I/O field_9" at 320,603 size 96x32; FormatPattern 999
      ProcessValue <- "Batch_Management_DB_PV_Lot_Status"
   IOField "I/O field_10" at 459,16 size 264x32; FormatPattern 999
      ProcessValue <- "Status_Batch_Number"
   IOField "I/O field_11" at 473,600 size 96x32; FormatPattern s99999
      ProcessValue <- "Batch_Management_DB_Record_Number"
   Button "Button_1" at 802,503 size 124x85; TextOff 'STop'
      on Press: StopRuntime(0)
   Button "Button_5" at 813,48 size 198x52; TextOff 'In lô'; TextList "Lot_Status"
      ObjectEnable <- "Hide"
      ProcessValue <- "Batch_Management_DB_PV_Lot_Status"
   TextField "Text field_3" at 824,14 size 177x29; Text 'Trạng thái lô'
   Rectangle "Rectangle_2" at 290,469 size 420x23
      Visibility <- "Batch_Management_DB_PV_Lot_Status"

VB script "Total_Blister"
   'Tip:
   ' 1. Use the <CTRL+SPACE> or <CTRL+I> shortcut to open a list of all objects and functions
   ' 2. Write the code using the HMI Runtime object.
   '  Example: HmiRuntime.Screens("Screen_1").
   ' 3. Use the <CTRL+J> shortcut to create an object reference.
   'Write the code as of this position:
   
   Dim Screen, WidthScreen, Blis(100), kc_2_cot, i, kc_hieudung,tongsocot,bung, letrai
   Dim cot
   SmartTags("Blister_Show_Total_Blister_Column") = SmartTags("Blister_Show_Total_Blister_Column_Temp")
   If SmartTags("Blister_Show_Total_Blister_Column") < 1 Then
   SmartTags("Blister_Show_Total_Blister_Column") = 1
   End If
   
   If SmartTags("Blister_Show_Total_Blister_Column") > 20 Then
   SmartTags("Blister_Show_Total_Blister_Column") = 20
   End If
   
   Set Screen = HmiRuntime.Screens("Blister_Setting")
   Set Blis(1) = HmiRuntime.Screens("Blister_Setting").ScreenItems("Blister_1")
   Set Blis(2) = HmiRuntime.Screens("Blister_Setting").ScreenItems("Blister_2")
   Set Blis(3) = HmiRuntime.Screens("Blister_Setting").ScreenItems("Blister_3")
   Set Blis(4) = HmiRuntime.Screens("Blister_Setting").ScreenItems("Blister_4")
   Set Blis(5) = HmiRuntime.Screens("Blister_Setting").ScreenItems("Blister_5")
   Set Blis(6) = HmiRuntime.Screens("Blister_Setting").ScreenItems("Blister_6")
   Set Blis(7) = HmiRuntime.Screens("Blister_Setting").ScreenItems("Blister_7")
   Set Blis(8) = HmiRuntime.Screens("Blister_Setting").ScreenItems("Blister_8")
   Set Blis(9) = HmiRuntime.Screens("Blister_Setting").ScreenItems("Blister_9")
   Set Blis(10) = HmiRuntime.Screens("Blister_Setting").ScreenItems("Blister_10")
   Set Blis(11) = HmiRuntime.Screens("Blister_Setting").ScreenItems("Blister_11")
   Set Blis(12) = HmiRuntime.Screens("Blister_Setting").ScreenItems("Blister_12")
   Set Blis(13) = HmiRuntime.Screens("Blister_Setting").ScreenItems("Blister_13")
   Set Blis(14) = HmiRuntime.Screens("Blister_Setting").ScreenItems("Blister_14")
   Set Blis(15) = HmiRuntime.Screens("Blister_Setting").ScreenItems("Blister_15")
   Set Blis(16) = HmiRuntime.Screens("Blister_Setting").ScreenItems("Blister_16")
   Set Blis(17) = HmiRuntime.Screens("Blister_Setting").ScreenItems("Blister_17")
   Set Blis(18) = HmiRuntime.Screens("Blister_Setting").ScreenItems("Blister_18")
   Set Blis(19) = HmiRuntime.Screens("Blister_Setting").ScreenItems("Blister_19")
   Set Blis(20) = HmiRuntime.Screens("Blister_Setting").ScreenItems("Blister_20")
   '-----------------------------
   
   For i = 1  To 20											' reset vi tri all vi
   Blis(i).left =  50
   Next
   '-----------------------------
   kc_hieudung = screen.Width - 200							'824
   tongsocot = SmartTags("Blister_Show_Total_Blister_Column")	
   '-------------------
   bung = tongsocot - 1
   If bung < 1 Then
   bung = 1
   End If
   '-------------------
   
   kc_2_cot = kc_hieudung/bung		
   
   cot = tongsocot
   
   If tongsocot > 1 Then
   letrai = 50	
   	
   For i = 2  To tongsocot
   cot = cot - 1
   letrai = letrai + kc_2_cot
   Blis(cot).left =  letrai 
   
   Next
   
   End If

VB script "Total_Blister_test"
   'Tip:
   ' 1. Use the <CTRL+SPACE> or <CTRL+I> shortcut to open a list of all objects and functions
   ' 2. Write the code using the HMI Runtime object.
   '  Example: HmiRuntime.Screens("Screen_1").
   ' 3. Use the <CTRL+J> shortcut to create an object reference.
   'Write the code as of this position:
   
   Dim Screen, WidthScreen, Blis(100), kc_2_cot, i, kc_hieudung,tongsocot,bung, letrai
   Dim cot, cycle,Do_rong_cot
   SmartTags("Blister_Show_Total_Blister_Column") = SmartTags("Blister_Show_Total_Blister_Column_Temp")
   If SmartTags("Blister_Show_Total_Blister_Column") < 1 Then
   SmartTags("Blister_Show_Total_Blister_Column") = 1
   End If
   
   If SmartTags("Blister_Show_Total_Blister_Column") > 20 Then
   SmartTags("Blister_Show_Total_Blister_Column") = 20
   End If
   
   Set Screen = HmiRuntime.Screens("Blister_Setting")
   Set Blis(1) = HmiRuntime.Screens("Blister_Setting").ScreenItems("Blister_1")
   Set Blis(2) = HmiRuntime.Screens("Blister_Setting").ScreenItems("Blister_2")
   Set Blis(3) = HmiRuntime.Screens("Blister_Setting").ScreenItems("Blister_3")
   Set Blis(4) = HmiRuntime.Screens("Blister_Setting").ScreenItems("Blister_4")
   Set Blis(5) = HmiRuntime.Screens("Blister_Setting").ScreenItems("Blister_5")
   Set Blis(6) = HmiRuntime.Screens("Blister_Setting").ScreenItems("Blister_6")
   Set Blis(7) = HmiRuntime.Screens("Blister_Setting").ScreenItems("Blister_7")
   Set Blis(8) = HmiRuntime.Screens("Blister_Setting").ScreenItems("Blister_8")
   Set Blis(9) = HmiRuntime.Screens("Blister_Setting").ScreenItems("Blister_9")
   Set Blis(10) = HmiRuntime.Screens("Blister_Setting").ScreenItems("Blister_10")
   Set Blis(11) = HmiRuntime.Screens("Blister_Setting").ScreenItems("Blister_11")
   Set Blis(12) = HmiRuntime.Screens("Blister_Setting").ScreenItems("Blister_12")
   Set Blis(13) = HmiRuntime.Screens("Blister_Setting").ScreenItems("Blister_13")
   Set Blis(14) = HmiRuntime.Screens("Blister_Setting").ScreenItems("Blister_14")
   Set Blis(15) = HmiRuntime.Screens("Blister_Setting").ScreenItems("Blister_15")
   Set Blis(16) = HmiRuntime.Screens("Blister_Setting").ScreenItems("Blister_16")
   Set Blis(17) = HmiRuntime.Screens("Blister_Setting").ScreenItems("Blister_17")
   Set Blis(18) = HmiRuntime.Screens("Blister_Setting").ScreenItems("Blister_18")
   Set Blis(19) = HmiRuntime.Screens("Blister_Setting").ScreenItems("Blister_19")
   Set Blis(20) = HmiRuntime.Screens("Blister_Setting").ScreenItems("Blister_20")
   '-----------------------------
   For i = 1  To 20											' reset vi tri all vi
   Blis(i).left =  50
   Next
   '-----------------------------
   'kc_hieudung = screen.Width - 200							'824
   kc_hieudung = 824	
   
